(* CODESYS project Vorlage_Visualisierung_Station1.project

Project tree, tasks and I/O mapping:
  SoftSPS : CODESYS Control Win V3 x64, 3S - Smart Software Solutions GmbH, version 3.5.16.40
    application Application
      libraries: Standard, 3.5.15.0 (System)
      task MainTask (cyclic, interval t#15ms, priority 10) calls PLC_PRG
      task VISU_TASK (cyclic, interval 15 ms, priority 0) calls VisuElems.Visu_Prg, vis_Ablauf, vis_Zuweisung
      global variables GVL
      visualisation Visualization
      program PLC_PRG [ST]
      function block FB_Automatik [SFC]: Step4_active, Step5_active, Step7_active, Step8_active, Step10_active, Step9_active, Step12_active, Step6_active, Step14_active, Step13_active, Step17_active, Step18_active, Step19_active, Step24_active, Step25_active, Step22_active, Step23_active
      function block FB_Initialisierung [SFC]: Step0_active, Step1_active, Step2_active, Step3_active, Step4_active, Step5_active, Step11_active, Step7_active, Step8_active, Init_active, Step10_active, Step6_active, Step13_active, Step14_active, Step15_active, Step16_active, Step18_active, Step20_active, Step22_active, Step19_active, Step21_active, Step23_active, Step17_active, Step18_active_0, Step19_active_0, Step20_active_0, Step21_active_0, Step22_active_0, Step23_active_0, Step24_active
  libraries: VisuSymbols, 3.5.10.0 (System)
  text list GlobalTextList
  program vis_Zuweisung [ST]
  data type Flasche
  program vis_Ablauf [ST]
  function block FB_Quit [FBD]
  function block FB_Blink [FBD]
  function block FB_Lamps [ST]
  function block FB_BottleIdentification [ST]
*)

// Flasche
TYPE Flasche :
STRUCT
	Gross		:BOOL;
	Weiss		:BOOL;
	PX			:INT;
	PY			:INT;
	Aktiv		:INT;
	Blockiert	:BOOL;
END_STRUCT
END_TYPE

// SoftSPS/Application/GVL
VAR_GLOBAL
	(*INPUT*)
	i_Abtransport_LT		:BOOL;
	i_Annahme_LT_Eingang	:BOOL;
	i_Annahme_VE_heraus		:BOOL;
	i_Annahme_VE_hinein		:BOOL;
	i_Auto					:BOOL;
	i_BEKenn_LS_mitte		:BOOL;
	i_BEKenn_LS_oben		:BOOL;
	i_BEKenn_LT_unten		:BOOL;
	i_Lager1_LT_Ausgang		:BOOL;
	i_Lager1_LT_Eingang		:BOOL;
	i_Lager1_VE_heraus		:BOOL;
	i_Lager1_VE_hinein		:BOOL;
	i_Lager2_LT_Ausgang		:BOOL;
	i_Lager2_LT_Eingang		:BOOL;
	i_Lager2_VE_heraus		:BOOL;
	i_Lager2_VE_hinein		:BOOL;
	i_Lager2_We_gerade		:BOOL;
	i_Lager2_We_kurve		:BOOL;
	i_Lager3_LT_Ausgang		:BOOL;
	i_Lager3_LT_Eingang		:BOOL;
	i_Lager3_VE_heraus		:BOOL;
	i_Lager3_VE_hinein		:BOOL;
	i_Lager3_We_gerade		:BOOL;
	i_Lager3_We_kurve		:BOOL;
	i_Lager4_LT_Ausgang		:BOOL;
	i_Lager4_LT_Eingang		:BOOL;
	i_Lager4_VE_heraus		:BOOL;
	i_Lager4_VE_hinein		:BOOL;
	i_Lager4_We_gerade		:BOOL;
	i_Lager4_We_kurve		:BOOL;
	i_Notaus				:BOOL;
	i_Quit					:BOOL;
	i_Rueckl_LT_Ausgang		:BOOL;
	i_Rueckl_LT_Eingang		:BOOL;
	i_Rueckl_VE_heraus		:BOOL;
	i_Rueckl_VE_hinein		:BOOL;
	i_Rueckl_We_gerade		:BOOL;
	i_Rueckl_We_kurve		:BOOL;
	i_Schritt				:BOOL;
	i_Weiter				:BOOL;
	(*OUTPUT*)		
	o_Annahme_Band			:BOOL;
	o_Annahme_VE			:BOOL;
	o_Auto					:BOOL;
	o_Fehler				:BOOL;
	o_Lager1_Band			:BOOL;
	o_Lager1_VE				:BOOL;
	o_Lager2_Band			:BOOL;
	o_Lager2_VE				:BOOL;
	o_Lager2_Weiche			:BOOL;
	o_Lager3_Band			:BOOL;
	o_Lager3_VE				:BOOL;
	o_Lager3_Weiche			:BOOL;
	o_Lager4_Band			:BOOL;
	o_Lager4_VE				:BOOL;
	o_Lager4_Weiche			:BOOL;
	o_Rueckl_Band			:BOOL;
	o_Rueckl_VE				:BOOL;
	o_Rueckl_Weiche			:BOOL;
	o_Sammelband_anaus		:BOOL;
	o_Sammelband_Richtung	:BOOL;
	o_Schritt				:BOOL;
	o_Status				:BOOL;
	o_Weichenband			:BOOL;		
END_VAR

// SoftSPS/Application/PLC_PRG
PROGRAM PLC_PRG
VAR
	fb_Quit	:FB_Quit;
	fb_Blink:FB_Blink;
	fb_Lamps:FB_Lamps;
	fb_Automatik: FB_Automatik;
	fb_Initialisierung:FB_Initialisierung;
	m_Idle:					BOOL;
	m_Init:					BOOL;
	m_Automatic:			BOOL;
	m_EmergencyOff:			BOOL;
	m_temp_InitSuccessful:	BOOL;
	m_Fehler:				BOOL;
END_VAR

fb_Quit(i_quittieren:=GVL.i_Quit);

IF NOT GVL.i_Notaus THEN
 m_EmergencyOff := 1;
 m_Idle := 0;
 m_Init := 0;
 m_Automatic := 0;
 m_temp_InitSuccessful:=0;
 
END_IF

IF m_Idle AND GVL.i_Schritt THEN
 m_Init := 1;
 m_Idle := 0;
 m_EmergencyOff :=0;
 m_Automatic :=0;
 fb_Initialisierung(SFCInit:=1);	
END_IF

IF m_Init AND NOT m_temp_InitSuccessful THEN
	fb_Initialisierung(SFCInit:=0);
	m_temp_InitSuccessful:=fb_Initialisierung.o_InitSuccessful;
END_IF

IF m_Init AND m_temp_InitSuccessful AND GVL.i_Auto THEN
 m_Automatic := 1;
 m_EmergencyOff :=0;
 m_Idle :=0;
 m_Init :=0;
END_IF

fb_Lamps(i_Idle:=m_Idle,i_Init:=m_Init,i_EmergencyOff:= m_EmergencyOff,i_Automatic:= m_Automatic,i_EmergencyOffButton:= GVL.i_Notaus,i_InitSuccessful:= m_temp_InitSuccessful,i_Fehler:=m_Fehler);

GVL.o_Status:=fb_Lamps.o_Status;
GVL.o_Fehler:=fb_Lamps.o_Fehler;
GVL.o_Auto:=fb_Lamps.o_Auto;
GVL.o_Schritt:=fb_Lamps.o_Schritt; 

IF m_EmergencyOff AND GVL.i_Notaus AND fb_Quit.o_quittieren THEN
 m_Idle := 1;
 m_EmergencyOff :=0;
 m_Init :=0;
 m_Automatic  :=0; 
 m_temp_InitSuccessful:=0;
END_IF



WHILE m_Automatic AND GVL.i_Notaus DO	
	fb_Automatik(SFCInit:=0);
END_WHILE

IF m_Automatic AND NOT GVL.i_Notaus THEN
	fb_Automatik(SFCInit:=1);
END_IF

END_PROGRAM

// FB_Quit
FUNCTION_BLOCK FB_Quit
VAR_INPUT
	i_quittieren: BOOL;
END_VAR
VAR_OUTPUT
	 o_quittieren: BOOL;
END_VAR
VAR
	f_trig_0: F_TRIG;
	ton_0: TON;
	tp_0: TP;
	tp_1: TP;
	TON_1: TON;
END_VAR

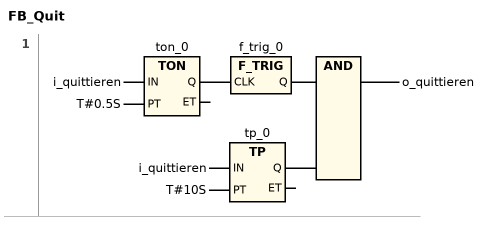
// NETWORK 1
ton_0(IN := i_quittieren, PT := T#0.5S); // TON
f_trig_0(CLK := ton_0.Q); // F_TRIG
tp_0(IN := i_quittieren, PT := T#10S); // TP
o_quittieren := f_trig_0.Q AND tp_0.Q;

END_FUNCTION_BLOCK

// SoftSPS/Application/FB_Initialisierung
FUNCTION_BLOCK FB_Initialisierung
VAR_INPUT
	SFCInit : BOOL;
END_VAR
VAR_OUTPUT
	o_InitSuccessful:BOOL;
END_VAR
VAR
	fb_BottleIdentification :FB_BottleIdentification;
	fb_Ton:Ton;
	h:INT;
	bottleType: INT;
	lagerFrei: BOOL;
	flascheAngekommen: BOOL;
END_VAR

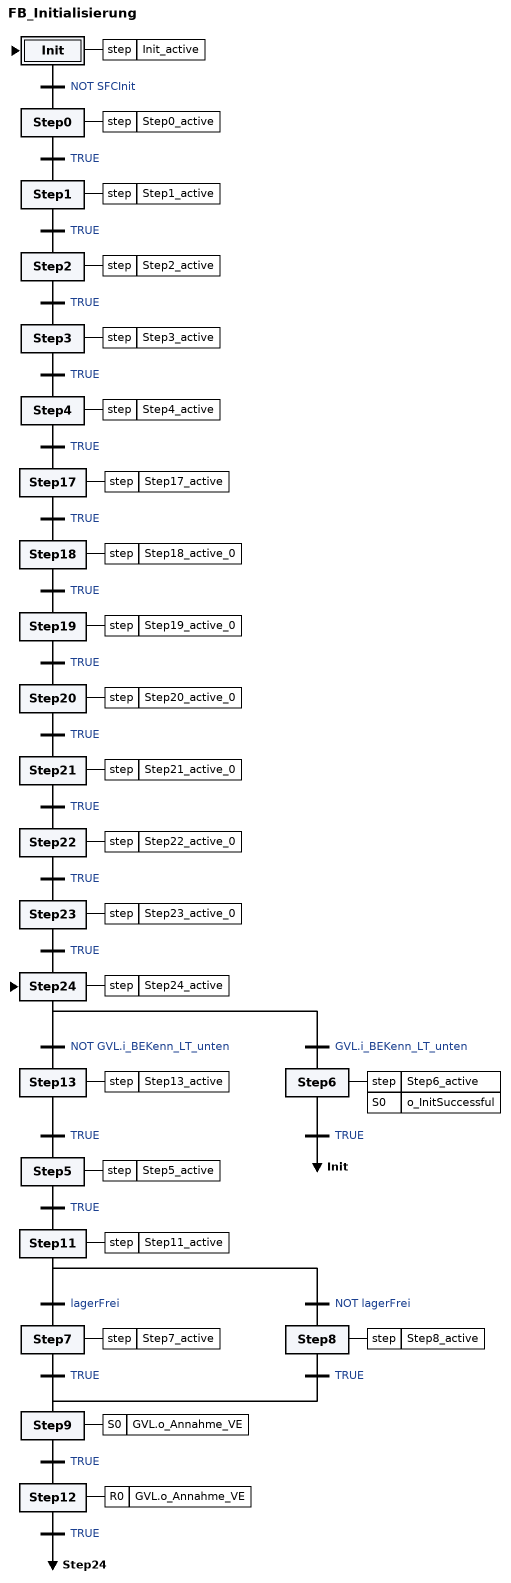
INITIAL_STEP Init:
    Init_active(N);  // step action
END_STEP
TRANSITION FROM Init TO Step0
    := NOT SFCInit;
END_TRANSITION
STEP Step0:
    Step0_active(N);  // step action
END_STEP
TRANSITION FROM Step0 TO Step1
    := TRUE;
END_TRANSITION
STEP Step1:  // min time T#1s
    Step1_active(N);  // step action
END_STEP
TRANSITION FROM Step1 TO Step2
    := TRUE;
END_TRANSITION
STEP Step2:  // min time T#1s
    Step2_active(N);  // step action
END_STEP
TRANSITION FROM Step2 TO Step3
    := TRUE;
END_TRANSITION
STEP Step3:  // min time T#1s
    Step3_active(N);  // step action
END_STEP
TRANSITION FROM Step3 TO Step4
    := TRUE;
END_TRANSITION
STEP Step4:  // min time T#2s
    Step4_active(N);  // step action
END_STEP
TRANSITION FROM Step4 TO Step17
    := TRUE;
END_TRANSITION
STEP Step17:  // min time T#1s
    Step17_active(N);  // step action
END_STEP
TRANSITION FROM Step17 TO Step18
    := TRUE;
END_TRANSITION
STEP Step18:  // min time T#1s
    Step18_active_0(N);  // step action
END_STEP
TRANSITION FROM Step18 TO Step19
    := TRUE;
END_TRANSITION
STEP Step19:  // min time T#1s
    Step19_active_0(N);  // step action
END_STEP
TRANSITION FROM Step19 TO Step20
    := TRUE;
END_TRANSITION
STEP Step20:  // min time T#1s
    Step20_active_0(N);  // step action
END_STEP
TRANSITION FROM Step20 TO Step21
    := TRUE;
END_TRANSITION
STEP Step21:  // min time T#1s
    Step21_active_0(N);  // step action
END_STEP
TRANSITION FROM Step21 TO Step22
    := TRUE;
END_TRANSITION
STEP Step22:  // min time T#1s
    Step22_active_0(N);  // step action
END_STEP
TRANSITION FROM Step22 TO Step23
    := TRUE;
END_TRANSITION
STEP Step23:  // min time T#1s
    Step23_active_0(N);  // step action
END_STEP
TRANSITION FROM Step23 TO Step24
    := TRUE;
END_TRANSITION
STEP Step24:  // min time T#10s
    Step24_active(N);  // step action
END_STEP
TRANSITION FROM Step24 TO Step13
    := NOT GVL.i_BEKenn_LT_unten;
END_TRANSITION
STEP Step13:
    Step13_active(N);  // step action
END_STEP
TRANSITION FROM Step13 TO Step5
    := TRUE;
END_TRANSITION
STEP Step5:
    Step5_active(N);  // step action
END_STEP
TRANSITION FROM Step5 TO Step11
    := TRUE;
END_TRANSITION
STEP Step11:
    Step11_active(N);  // step action
END_STEP
TRANSITION FROM Step11 TO Step7
    := lagerFrei;
END_TRANSITION
STEP Step7:
    Step7_active(N);  // step action
END_STEP
TRANSITION FROM Step7 TO Step9
    := TRUE;
END_TRANSITION
TRANSITION FROM Step11 TO Step8
    := NOT lagerFrei;
END_TRANSITION
STEP Step8:
    Step8_active(N);  // step action
END_STEP
TRANSITION FROM Step8 TO Step9
    := TRUE;
END_TRANSITION
STEP Step9:  // min time T#2s
    GVL.o_Annahme_VE(S0);
END_STEP
TRANSITION FROM Step9 TO Step12
    := TRUE;
END_TRANSITION
STEP Step12:  // min time T#5s
    GVL.o_Annahme_VE(R0);
END_STEP
TRANSITION FROM Step12 TO Step24
    := TRUE;
END_TRANSITION
TRANSITION FROM Step24 TO Step6
    := GVL.i_BEKenn_LT_unten;
END_TRANSITION
STEP Step6:
    Step6_active(N);  // step action
    o_InitSuccessful(S0);
END_STEP
TRANSITION FROM Step6 TO Init
    := TRUE;
END_TRANSITION

ACTION Step0_active:
GVL.o_Annahme_VE:=0;
GVL.o_Lager1_VE:=1;
GVL.o_Lager2_VE:=1;
GVL.o_Lager3_VE:=1;
GVL.o_Lager4_VE:=1;
GVl.o_Rueckl_VE:=1;
GVL.o_Weichenband:=1;
END_ACTION

ACTION Step1_active:
GVL.o_Annahme_Band:=1;
GVL.o_Rueckl_Band:=1;
GVL.o_Rueckl_VE:=1;
END_ACTION

ACTION Step2_active:
GVL.o_Lager3_Band:=1;
GVL.o_Lager4_Band:=1;
END_ACTION

ACTION Step3_active:
GVL.o_Lager1_Band:=1;
GVL.o_Lager2_Band:=1;
END_ACTION

ACTION Step4_active:
GVL.o_Sammelband_anaus:=1;
GVL.o_Sammelband_Richtung:=1;
END_ACTION

ACTION Step5_active:
fb_BottleIdentification(i_LS_Top:=GVL.i_BEKenn_LS_oben, i_LS_Middle:=GVL.i_BEKenn_LS_mitte);
bottleType:=fb_BottleIdentification.o_BottleType;
END_ACTION

ACTION Step11_active:
CASE bottleType OF
	1: 	IF GVL.i_Lager1_LT_Eingang THEN
			lagerFrei:=1;
		ELSE
			lagerFrei:=0;	
		END_IF
	2: 	IF GVL.i_Lager2_LT_Eingang THEN
			lagerFrei:=1;
		ELSE
			lagerFrei:=0;	
		END_IF
	3: 	IF GVL.i_Lager3_LT_Eingang THEN
			lagerFrei:=1;
		ELSE
			lagerFrei:=0;	
		END_IF
	4: 	IF GVL.i_Lager4_LT_Eingang THEN
			lagerFrei:=1;
		ELSE
			lagerFrei:=0;	
		END_IF
END_CASE
END_ACTION

ACTION Step7_active:
CASE bottleType OF
	
	2: GVL.o_Lager2_Weiche:=1;
	3: GVL.o_Lager3_Weiche:=1;	
	4: GVL.o_Lager4_Weiche:=1;	

END_CASE
END_ACTION

ACTION Step8_active:
GVL.o_Rueckl_Weiche:=1;
END_ACTION

ACTION Init_active:
IF SFCInit THEN
	GVL.o_Lager1_Band:=0;
	GVL.o_Lager1_Band:=0;
	GVL.o_Lager1_Band:=0;
	GVL.o_Lager1_Band:=0;
	GVL.o_Annahme_Band:=0;
	GVL.o_Rueckl_Band:=0;
	GVL.o_Weichenband:=0;
	GVL.o_Sammelband_anaus:=0;
	
END_IF
END_ACTION

ACTION Step10_active:

END_ACTION

ACTION Step6_active:
GVL.o_Lager2_Weiche:=0;
GVL.o_Lager3_Weiche:=0;
GVL.o_Lager4_Weiche:=0;
GVL.o_Rueckl_Weiche:=0;

GVL.o_Annahme_Band:=0;
GVL.o_Rueckl_Band:=0;
GVL.o_Lager3_Band:=0;
GVL.o_Lager4_Band:=0;
GVL.o_Lager1_Band:=0;
GVL.o_Lager2_Band:=0;
GVL.o_Sammelband_anaus:=0;
END_ACTION

ACTION Step13_active:
GVL.o_Lager2_Weiche:=0;
GVL.o_Lager3_Weiche:=0;
GVL.o_Lager4_Weiche:=0;
GVL.o_Rueckl_Weiche:=0;
END_ACTION

ACTION Step14_active:
// NETWORK 1
END_ACTION

ACTION Step15_active:
GVL.o_Rueckl_VE:=0;
END_ACTION

ACTION Step16_active:
GVL.o_Rueckl_VE:=1;
END_ACTION

ACTION Step18_active:
GVL.o_Rueckl_VE:=0;
END_ACTION

ACTION Step20_active:

END_ACTION

ACTION Step22_active:
GVL.o_Rueckl_VE:=0;
END_ACTION

ACTION Step19_active:
GVL.o_Rueckl_VE:=1;
END_ACTION

ACTION Step21_active:
GVL.o_Rueckl_VE:=1;
END_ACTION

ACTION Step23_active:
GVL.o_Rueckl_VE:=1;
END_ACTION

ACTION Step17_active:
GVL.o_Rueckl_VE :=0;
END_ACTION

ACTION Step18_active_0:
GVL.o_Rueckl_VE :=1;
END_ACTION

ACTION Step19_active_0:
GVL.o_Rueckl_VE :=0;
END_ACTION

ACTION Step20_active_0:
GVL.o_Rueckl_VE :=1;
END_ACTION

ACTION Step21_active_0:
GVL.o_Rueckl_VE :=0;
END_ACTION

ACTION Step22_active_0:
GVL.o_Rueckl_VE :=1;
END_ACTION

ACTION Step23_active_0:
GVL.o_Rueckl_VE :=0;
END_ACTION

ACTION Step24_active:
GVL.o_Rueckl_VE :=1;
END_ACTION

END_FUNCTION_BLOCK

// FB_BottleIdentification
FUNCTION_BLOCK FB_BottleIdentification
VAR_INPUT
i_LS_Top: BOOL;
i_LS_Middle: BOOL;
END_VAR
VAR_OUTPUT
o_BottleType: INT;
END_VAR
VAR
END_VAR

IF i_LS_Top AND i_LS_Middle THEN
 o_BottleType:=1;
ELSIF NOT i_LS_Top AND i_LS_Middle THEN
 o_BottleType:=2;
ELSIF i_LS_Top AND NOT i_LS_Middle THEN
 o_BottleType:=3;
ELSE
 o_BottleType:=4;
END_IF

END_FUNCTION_BLOCK

// FB_Lamps
FUNCTION_BLOCK FB_Lamps
VAR_INPUT
	 i_Idle: BOOL;
	 i_Init: BOOL;
	 i_Fehler: BOOL;
	 i_EmergencyOff: BOOL;
	 i_Automatic: BOOL;
	 i_EmergencyOffButton: BOOL;
	 i_InitSuccessful: BOOL;
     
END_VAR
VAR_OUTPUT
	 o_Status: BOOL;
     o_Fehler: BOOL;
	 o_Auto: BOOL;
	 o_Schritt: BOOL;
END_VAR
VAR
	fb_Blink: FB_Blink;
END_VAR

IF i_Idle  AND NOT i_Automatic THEN
 fb_Blink(i_BlinkTime:=T#1S);
 o_Status:=fb_Blink.o_Blink;
ELSIF NOT i_Idle  AND i_Automatic THEN
 o_Status:=   1;
 o_Auto:=   1;
 o_Schritt:=   0;
ELSIF i_Init AND NOT i_InitSuccessful THEN
 fb_Blink(i_BlinkTime:=T#500MS);
 o_Status:=     1;
 o_Schritt:=fb_Blink.o_Blink;
 
ELSIF i_Init AND i_InitSuccessful THEN
 o_Status:=   1;
  o_Schritt:=   1;
ELSE
 o_Status:=   0;
 o_Auto:=   0;
 o_Schritt:=   0;
END_IF


IF  i_EmergencyOffButton AND i_EmergencyOff AND NOT i_Fehler THEN
 fb_Blink(i_BlinkTime:=T#167MS);
 o_Fehler:=fb_Blink.o_Blink;
ELSIF i_Fehler OR i_EmergencyOff THEN
 o_Fehler:=   1;
ELSE 
 o_Fehler:=   0;
END_IF

END_FUNCTION_BLOCK

// FB_Blink
FUNCTION_BLOCK FB_Blink
VAR_INPUT
	i_BlinkTime: TIME;
END_VAR
VAR_OUTPUT
	o_Blink: BOOL;
END_VAR
VAR
	ton0: TON;
	ton1: TON;
END_VAR

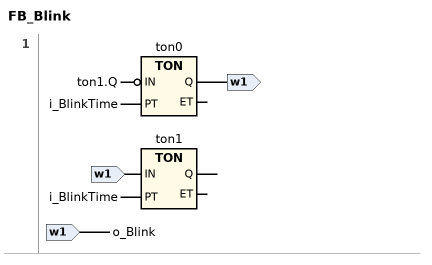
// NETWORK 1
ton0(IN := NOT ton1.Q, PT := i_BlinkTime); // TON
ton1(IN := ton0.Q, PT := i_BlinkTime); // TON
o_Blink := ton0.Q;

END_FUNCTION_BLOCK

// SoftSPS/Application/FB_Automatik
FUNCTION_BLOCK FB_Automatik
VAR_INPUT
	SFCInit : BOOL;
END_VAR
VAR_OUTPUT
END_VAR
VAR
	counter :INT;
	lagerFrei: BOOL;
	fb_BottleIdentification :FB_BottleIdentification;
	bottleType: INT;
	flascheAngekommen: BOOL;
	Timer: BOOL;
	flascheAnLager: BOOL;
END_VAR

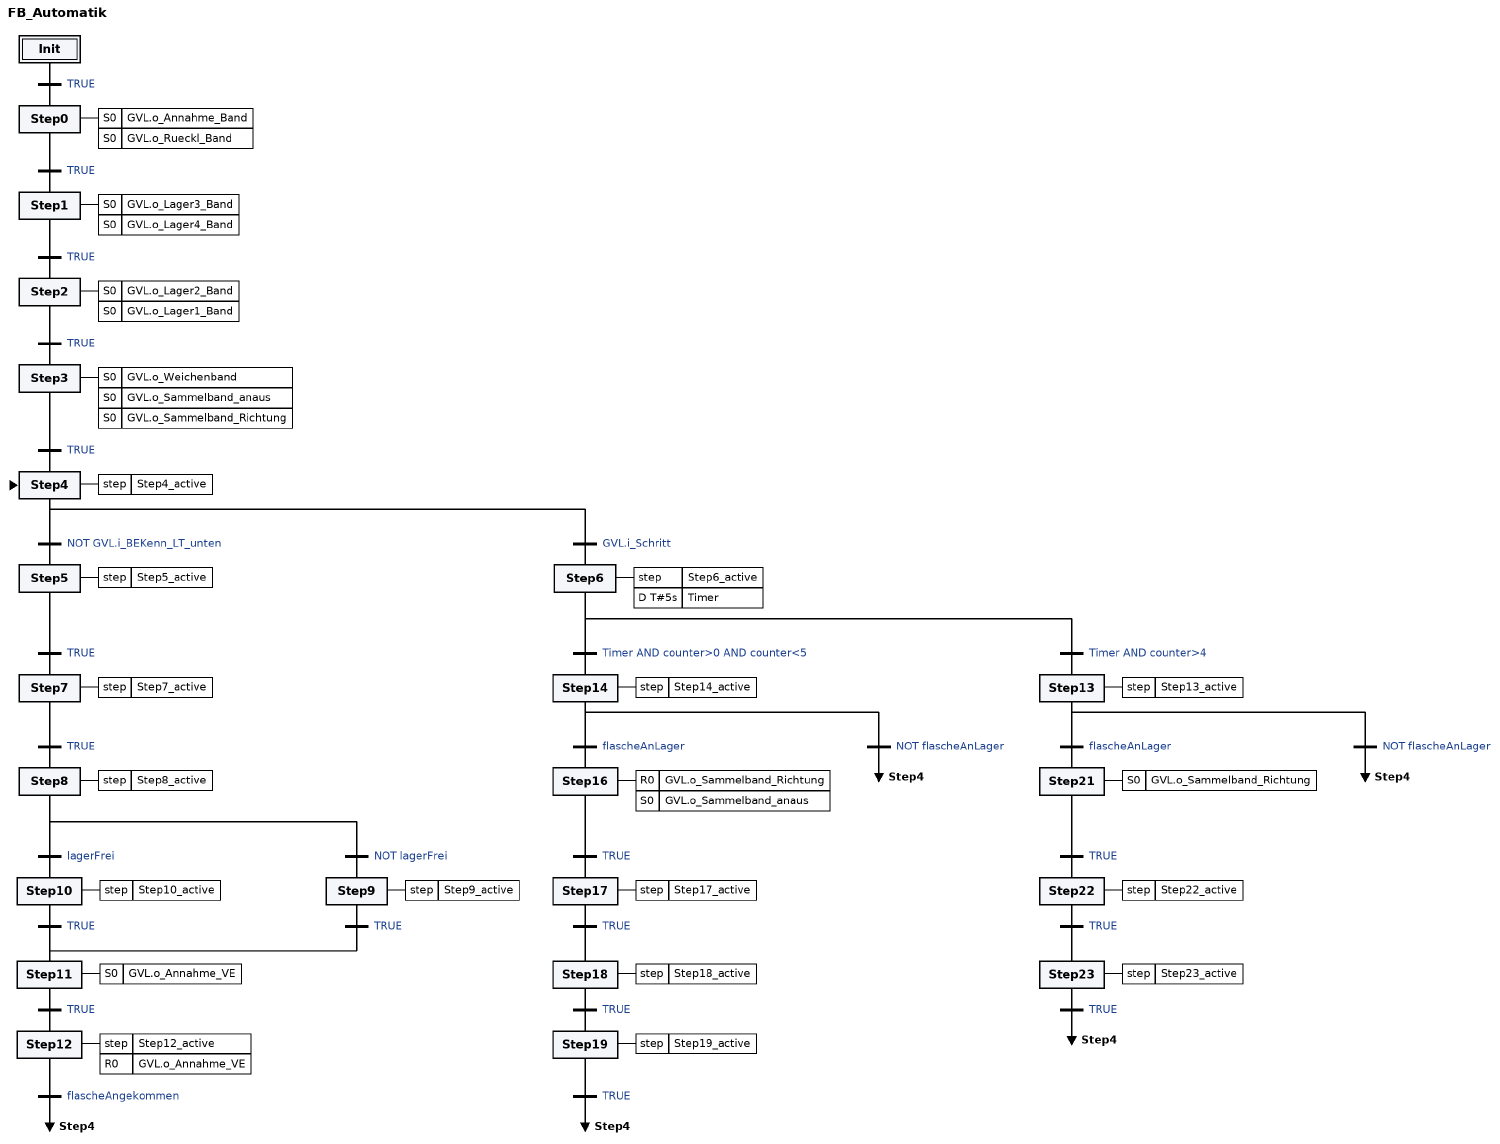
INITIAL_STEP Init:
END_STEP
TRANSITION FROM Init TO Step0
    := TRUE;
END_TRANSITION
STEP Step0:  // min time T#1s
    GVL.o_Annahme_Band(S0);
    GVL.o_Rueckl_Band(S0);
END_STEP
TRANSITION FROM Step0 TO Step1
    := TRUE;
END_TRANSITION
STEP Step1:  // min time T#1s
    GVL.o_Lager3_Band(S0);
    GVL.o_Lager4_Band(S0);
END_STEP
TRANSITION FROM Step1 TO Step2
    := TRUE;
END_TRANSITION
STEP Step2:  // min time T#1s
    GVL.o_Lager2_Band(S0);
    GVL.o_Lager1_Band(S0);
END_STEP
TRANSITION FROM Step2 TO Step3
    := TRUE;
END_TRANSITION
STEP Step3:
    GVL.o_Weichenband(S0);
    GVL.o_Sammelband_anaus(S0);
    GVL.o_Sammelband_Richtung(S0);
END_STEP
TRANSITION FROM Step3 TO Step4
    := TRUE;
END_TRANSITION
STEP Step4:
    Step4_active(N);  // step action
END_STEP
TRANSITION FROM Step4 TO Step5
    := NOT GVL.i_BEKenn_LT_unten;
END_TRANSITION
STEP Step5:
    Step5_active(N);  // step action
END_STEP
TRANSITION FROM Step5 TO Step7
    := TRUE;
END_TRANSITION
STEP Step7:
    Step7_active(N);  // step action
END_STEP
TRANSITION FROM Step7 TO Step8
    := TRUE;
END_TRANSITION
STEP Step8:
    Step8_active(N);  // step action
END_STEP
TRANSITION FROM Step8 TO Step10
    := lagerFrei;
END_TRANSITION
STEP Step10:
    Step10_active(N);  // step action
END_STEP
TRANSITION FROM Step10 TO Step11
    := TRUE;
END_TRANSITION
TRANSITION FROM Step8 TO Step9
    := NOT lagerFrei;
END_TRANSITION
STEP Step9:
    Step9_active(N);  // step action
END_STEP
TRANSITION FROM Step9 TO Step11
    := TRUE;
END_TRANSITION
STEP Step11:  // min time t#2s
    GVL.o_Annahme_VE(S0);
END_STEP
TRANSITION FROM Step11 TO Step12
    := TRUE;
END_TRANSITION
STEP Step12:  // min time T#8s
    Step12_active(N);  // step action
    GVL.o_Annahme_VE(R0);
END_STEP
TRANSITION FROM Step12 TO Step4
    := flascheAngekommen;
END_TRANSITION
TRANSITION FROM Step4 TO Step6
    := GVL.i_Schritt;
END_TRANSITION
STEP Step6:
    Step6_active(N);  // step action
    Timer(D, T#5s);
END_STEP
TRANSITION FROM Step6 TO Step14
    := Timer AND counter>0 AND counter<5;
END_TRANSITION
STEP Step14:
    Step14_active(N);  // step action
END_STEP
TRANSITION FROM Step14 TO Step16
    := flascheAnLager;
END_TRANSITION
STEP Step16:
    GVL.o_Sammelband_Richtung(R0);
    GVL.o_Sammelband_anaus(S0);
END_STEP
TRANSITION FROM Step16 TO Step17
    := TRUE;
END_TRANSITION
STEP Step17:  // min time T#2s
    Step17_active(N);  // step action
END_STEP
TRANSITION FROM Step17 TO Step18
    := TRUE;
END_TRANSITION
STEP Step18:  // min time t#2s
    Step18_active(N);  // step action
END_STEP
TRANSITION FROM Step18 TO Step19
    := TRUE;
END_TRANSITION
STEP Step19:
    Step19_active(N);  // step action
END_STEP
TRANSITION FROM Step19 TO Step4
    := TRUE;
END_TRANSITION
TRANSITION FROM Step14 TO Step4
    := NOT flascheAnLager;
END_TRANSITION
TRANSITION FROM Step6 TO Step13
    := Timer AND counter>4;
END_TRANSITION
STEP Step13:
    Step13_active(N);  // step action
END_STEP
TRANSITION FROM Step13 TO Step21
    := flascheAnLager;
END_TRANSITION
STEP Step21:
    GVL.o_Sammelband_Richtung(S0);
END_STEP
TRANSITION FROM Step21 TO Step22
    := TRUE;
END_TRANSITION
STEP Step22:  // min time t#2s
    Step22_active(N);  // step action
END_STEP
TRANSITION FROM Step22 TO Step23
    := TRUE;
END_TRANSITION
STEP Step23:
    Step23_active(N);  // step action
END_STEP
TRANSITION FROM Step23 TO Step4
    := TRUE;
END_TRANSITION
TRANSITION FROM Step13 TO Step4
    := NOT flascheAnLager;
END_TRANSITION

ACTION Step4_active:
GVL.o_Lager1_VE:=1;
GVL.o_Lager2_VE:=1;
GVL.o_Lager3_VE:=1;
GVL.o_Lager4_VE:=1;

counter:=0;
END_ACTION

ACTION Step5_active:
GVL.o_Lager2_Weiche:=0;
GVL.o_Lager3_Weiche:=0;
GVL.o_Lager4_Weiche:=0;
GVL.o_Rueckl_Weiche:=0;
END_ACTION

ACTION Step7_active:
fb_BottleIdentification(i_LS_Top:=GVL.i_BEKenn_LS_oben, i_LS_Middle:=GVL.i_BEKenn_LS_mitte);
bottleType:=fb_BottleIdentification.o_BottleType;
END_ACTION

ACTION Step8_active:
CASE bottleType OF
	1: 	IF GVL.i_Lager1_LT_Eingang THEN
			lagerFrei:=1;
		ELSE
			lagerFrei:=0;	
		END_IF
	2: 	IF GVL.i_Lager2_LT_Eingang THEN
			lagerFrei:=1;
		ELSE
			lagerFrei:=0;	
		END_IF
	3: 	IF GVL.i_Lager3_LT_Eingang THEN
			lagerFrei:=1;
		ELSE
			lagerFrei:=0;	
		END_IF
	4: 	IF GVL.i_Lager4_LT_Eingang THEN
			lagerFrei:=1;
		ELSE
			lagerFrei:=0;	
		END_IF
END_CASE
END_ACTION

ACTION Step10_active:
CASE bottleType OF
	
	2: GVL.o_Lager2_Weiche:=1;
	3: GVL.o_Lager3_Weiche:=1;	
	4: GVL.o_Lager4_Weiche:=1;	

END_CASE
END_ACTION

ACTION Step9_active:
GVL.o_Rueckl_Weiche:=1;
END_ACTION

ACTION Step12_active:
CASE bottleType OF
	1: 	IF NOT GVL.i_Lager1_LT_Eingang THEN
			flascheAngekommen:=1;
		END_IF
	2: 	IF NOT GVL.i_Lager2_LT_Eingang THEN
			flascheAngekommen:=1;
			
		END_IF
	3:  IF NOT GVL.i_Lager3_LT_Eingang THEN
			flascheAngekommen:=1;
			
		END_IF
	4:  IF NOT GVL.i_Lager4_LT_Eingang THEN
			flascheAngekommen:=1;
			
		END_IF
				
END_CASE
END_ACTION

ACTION Step6_active:
IF i_Schritt THEN
	
	WHILE i_Schritt DO
		counter := counter;
	END_WHILE
	
	counter :=counter+1;
END_IF
END_ACTION

ACTION Step14_active:
CASE counter OF
	
	1: 	IF GVL.i_Lager1_LT_Ausgang THEN
			flascheAnLager :=0;
		ELSE
			flascheAnLager :=1;
		END_IF
	2:  IF GVL.i_Lager2_LT_Ausgang THEN
			flascheAnLager :=0;
		ELSE
			flascheAnLager :=1;			
		END_IF
	3:  IF GVL.i_Lager3_LT_Ausgang THEN
			flascheAnLager :=0;
		ELSE
			flascheAnLager :=1;			
		END_IF
	4:  IF GVL.i_Lager4_LT_Ausgang THEN
			flascheAnLager :=0;
		ELSE
			flascheAnLager :=1;			
		END_IF
		
END_CASE
END_ACTION

ACTION Step13_active:
IF GVL.i_Rueckl_LT_Ausgang THEN
		flascheAnLager :=0;
ELSE
		flascheAnLager :=1;
END_IF
END_ACTION

ACTION Step17_active:
CASE counter OF
	
	1: 	GVL.o_Lager1_VE:=0;
	2:  GVL.o_Lager2_VE:=0;
	3:  GVL.o_Lager3_VE:=0;
	4:  GVL.o_Lager4_VE:=0;
		
END_CASE
END_ACTION

ACTION Step18_active:
CASE counter OF
	
	1: 	GVL.o_Lager1_VE:=1;
	2:  GVL.o_Lager2_VE:=1;
	3:  GVL.o_Lager3_VE:=1;
	4:  GVL.o_Lager4_VE:=1;
		
END_CASE
END_ACTION

ACTION Step19_active:
CASE counter OF
	
	1: 	GVL.o_Lager1_VE:=0;
	2:  GVL.o_Lager2_VE:=0;
	3:  GVL.o_Lager3_VE:=0;
	4:  GVL.o_Lager4_VE:=0;
		
END_CASE
END_ACTION

ACTION Step24_active:
GVL.o_Rueckl_VE :=0;
END_ACTION

ACTION Step25_active:
GVL.o_Rueckl_VE :=1;
END_ACTION

ACTION Step22_active:
GVL.o_Rueckl_VE :=0;
END_ACTION

ACTION Step23_active:
GVL.o_Rueckl_VE :=1;
END_ACTION

END_FUNCTION_BLOCK

// vis_Ablauf
PROGRAM vis_Ablauf
VAR_INPUT 
	Flaschen			:ARRAY [1..50] OF Flasche;
	Taster_Flasche		:ARRAY [1..50] OF BOOL;
	Anlageanaus			:BOOL;
END_VAR

VAR
	i_aktuell		:INT;
	i_Zaehler		:INT;
	i_aktuell_x		:INT;
	i_aktuell_y		:INT;
	Merker_Blockiert	:BOOL;
	
	Pixelpro2Zyklen: INT;
	Zyklus: 		INT;
	initial: 		INT;
	Zykluszaehler: 	INT;
	Merker_AB_LTE	:BOOL;
	Merker_FE_LSU	:BOOL;
	Merker_FE_LSM	:BOOL;
	Merker_FE_LSO	:BOOL;
	Merker_RL_LTE	:BOOL;
	Merker_RL_LTA	:BOOL;
	Merler_L1_LTE	:BOOL;
	Merler_L1_LTA	:BOOL;
	Merler_L2_LTE	:BOOL;
	Merler_L2_LTA	:BOOL;
	Merler_L3_LTE	:BOOL;
	Merler_L3_LTA	:BOOL;
	Merler_L4_LTE	:BOOL;
	Merler_L4_LTA	:BOOL;
	
	i_Zaehler2: 	INT;
	i_Zaehler3: 	INT;
	Startplatz_blockiert: BOOL;
	iInitial: 		INT := 1;
	i_Zaehler4: 	INT;
	Merker_AT_LT: 	BOOL;
	Merker_A5_CB:	BOOL;
	A5_CB_FF	:f_trig;
	A5_CB_RF	:r_trig;
	m_Init_Testcase	:BOOL;
	m_Init_Testcase_einmal :BOOL :=TRUE;
	M_Init_Stellung: BOOL;
	M_Init_Stellung_speicher: BOOL;
	i: INT;
END_VAR

Pixelpro2Zyklen := 1;
Zykluszaehler := Zykluszaehler +1;
IF Zykluszaehler = 1 THEN Zyklus := 1; Zykluszaehler := 0; ELSE Zyklus := 0; END_IF
IF iInitial = 1 THEN
	FOR i_Zaehler4 := 1 TO 50 DO
		IF i_Zaehler4 < 10 THEN Flaschen[i_Zaehler4].Gross := 0; Flaschen[i_Zaehler4].Weiss := 1; END_IF
		IF i_Zaehler4 >= 10 AND i_Zaehler4 < 20 THEN Flaschen[i_Zaehler4].Gross := 1; Flaschen[i_Zaehler4].Weiss := 1; END_IF
		IF i_Zaehler4 >= 20 AND i_Zaehler4 < 30 THEN Flaschen[i_Zaehler4].Gross := 0; Flaschen[i_Zaehler4].Weiss := 0; END_IF
		IF i_Zaehler4 >= 30 AND i_Zaehler4 < 40 THEN Flaschen[i_Zaehler4].Gross := 1; Flaschen[i_Zaehler4].Weiss := 0; END_IF
	END_FOR
	iInitial := 0;
END_IF

IF M_Init_Stellung = TRUE THEN //Einmalige Ausführung
	M_Init_Stellung_speicher:=TRUE;
	
	vis_Zuweisung.vis_o_Lager1_VE			:= TRUE;
	vis_Zuweisung.vis_o_Lager2_VE			:= TRUE;
	vis_Zuweisung.vis_o_Lager3_VE			:= TRUE;
	vis_Zuweisung.vis_o_Lager4_VE			:= TRUE;
	vis_Zuweisung.vis_o_Rueckl_VE			:= TRUE;
	GVL.o_Lager1_VE							:= TRUE;
	GVL.o_Lager2_VE							:= TRUE;
	GVL.o_Lager3_VE							:= TRUE;
	GVL.o_Lager4_VE							:= TRUE;
	GVL.o_Rueckl_VE							:= TRUE;
	GVL.o_Lager2_Weiche 					:= FALSE;
	GVL.o_Lager3_Weiche 					:= FALSE;
	GVL.o_Lager4_Weiche 					:= FALSE;
	GVL.o_Rueckl_Weiche 					:= FALSE;
	
	FOR i := 1 TO 50 DO
		Flaschen[i].Aktiv := 0;
		Flaschen[i].PX := 0;
		Flaschen[i].PY := 0 ;
	END_FOR
	
END_IF

IF M_Init_Stellung_speicher = TRUE THEN //Dauerhafte Ausführung bis Initialisierte Stellung eingenommen übernimmt
	
	IF TRUE THEN
			M_Init_Stellung_speicher := FALSE;
	END_IF
END_IF


IF m_Init_Testcase_einmal = TRUE AND m_Init_Testcase = TRUE THEN
	Flaschen[5].Aktiv := 1;
	Flaschen[5].PX := Flaschen[5].PX + 50;
	Flaschen[5].PY := Flaschen[5].PY ;
	Flaschen[11].Aktiv := 1;
	Flaschen[11].PX := Flaschen[11].PX + 350;
	Flaschen[11].PY := Flaschen[11].PY -90;
	Flaschen[14].Aktiv := 1;
	Flaschen[14].PX := Flaschen[14].PX + 30;
	Flaschen[14].PY := Flaschen[14].PY -390;
	Flaschen[23].Aktiv := 1;
	Flaschen[23].PX := Flaschen[23].PX + 190;
	Flaschen[23].PY := Flaschen[23].PY -90;
	Flaschen[36].Aktiv := 1;
	Flaschen[36].PX := Flaschen[36].PX + 580;
	Flaschen[36].PY := Flaschen[36].PY -200;
	GVL.o_Lager2_Weiche := TRUE;
	vis_Zuweisung.Lager2_Weiche_rot := -55;
	
	
	
	m_Init_Testcase_einmal := FALSE;
END_IF

  
FOR i_Zaehler3 := 1 TO 50 DO
	IF Flaschen[i_Zaehler3].PX <= 50 AND Flaschen[i_Zaehler3].PY = 0 AND Flaschen[i_Zaehler3].Aktiv = 1 THEN Startplatz_blockiert := 1; i_Zaehler3 := 51;
	ELSIF  Merker_A5_CB AND Flaschen[i_Zaehler3].PX <= 350 AND Flaschen[i_Zaehler3].PY = 0 AND Flaschen[i_Zaehler3].Aktiv = 1 THEN Startplatz_blockiert := 1; i_Zaehler3 := 51;
	ELSE Startplatz_blockiert := 0;
	END_IF
END_FOR


FOR i_Zaehler := 1 TO 50 DO
	
IF Taster_Flasche[i_Zaehler] = 1 AND Startplatz_blockiert = 0  THEN Flaschen[i_Zaehler].Aktiv := 1; END_IF

i_aktuell := i_Zaehler;
IF Flaschen[i_aktuell].Aktiv = 1 THEN
	
	i_aktuell_x := Flaschen[i_aktuell].PX;
	i_aktuell_y := Flaschen[i_aktuell].PY;
	

IF Flaschen[i_aktuell].Blockiert = 0 THEN
// Fahren
	
	// Fahren auf Annahmeband
		IF vis_Zuweisung.vis_o_Annahme_Band = 1 AND i_aktuell_y = 0 AND i_aktuell_x >= 0 AND i_aktuell_x < 580 THEN
			i_aktuell_x := i_aktuell_x +  Zyklus*Pixelpro2Zyklen; 
		END_IF
			
	// Fahren auf Rücklaufband
		IF vis_Zuweisung.vis_o_Rueckl_Band = 1 AND i_aktuell_y = -90 AND
		((i_aktuell_x = 580 AND vis_Zuweisung.vis_i_Rueckl_We_kurve = 1) OR (i_aktuell_x > 30 AND i_aktuell_x < 580)) THEN
			i_aktuell_x := i_aktuell_x -  Zyklus*Pixelpro2Zyklen; 
		END_IF
		
	// Fahren in Lager 4
		IF vis_Zuweisung.vis_o_Lager4_Band = 1 AND i_aktuell_y = -190 AND
		((i_aktuell_x = 580 AND vis_Zuweisung.vis_i_Lager4_We_kurve = 1 ) OR (i_aktuell_x > 30 AND i_aktuell_x < 580)) THEN
			i_aktuell_x := i_aktuell_x -  Zyklus*Pixelpro2Zyklen; 
		END_IF
		
	// Fahren in Lager 3
		IF vis_Zuweisung.vis_o_Lager3_Band = 1 AND i_aktuell_y = -290 AND
		((i_aktuell_x = 580 AND vis_Zuweisung.vis_i_Lager3_We_kurve = 1) OR (i_aktuell_x > 30 AND i_aktuell_x < 580)) THEN
			i_aktuell_x := i_aktuell_x -  Zyklus*Pixelpro2Zyklen; 
		END_IF
		
	// Fahren in Lager 2
		IF vis_Zuweisung.vis_o_Lager2_Band = 1 AND i_aktuell_y = -390 AND
		((i_aktuell_x = 580 AND vis_Zuweisung.vis_i_Lager2_We_kurve = 1) OR (i_aktuell_x > 30 AND i_aktuell_x < 580)) THEN
			i_aktuell_x := i_aktuell_x -  Zyklus*Pixelpro2Zyklen; 
		END_IF
		
	// Fahren in Lager 1
		IF vis_Zuweisung.vis_o_Lager1_Band = 1 AND i_aktuell_y = -490 AND i_aktuell_x >= -100 AND i_aktuell_x < 581 THEN
			i_aktuell_x := i_aktuell_x -  Zyklus*Pixelpro2Zyklen; 
		END_IF
		
	// Fahren auf Weichenband
		IF vis_Zuweisung.vis_o_Weichenband = 1 AND i_aktuell_x = 580 AND i_aktuell_y <= 0 AND i_aktuell_y > -490 THEN
			i_aktuell_y := i_aktuell_y -  Zyklus*Pixelpro2Zyklen; 
		END_IF
		
	// Fahren auf Sammelband
		IF vis_Zuweisung.vis_o_Sammelband_anaus = 1 AND i_aktuell_x = 30 AND i_aktuell_y < 0 AND i_aktuell_y > -490 THEN
		IF vis_Zuweisung.vis_o_Sammelband_Richtung = 1 THEN i_aktuell_y := i_aktuell_y +  Zyklus*Pixelpro2Zyklen; END_IF
		IF vis_Zuweisung.vis_o_Sammelband_Richtung = 0 THEN i_aktuell_y := i_aktuell_y -  Zyklus*Pixelpro2Zyklen; END_IF
		END_IF
	
			
		
END_IF

		
// Blockieren durch Weichen und Vereinzeler

		Merker_Blockiert := 0;
// Weichen auf Weichenband
	
	// Weiche Rücklauf
		IF i_aktuell_x = 580 AND i_aktuell_y = -90 AND vis_Zuweisung.vis_i_Rueckl_We_kurve = 1 AND vis_Zuweisung.vis_o_Rueckl_Band = 0 THEN 
		Flaschen[i_aktuell].Blockiert := 1; Merker_Blockiert := 1;
		ELSIF i_aktuell_x = 580 AND i_aktuell_y = -90 AND (vis_Zuweisung.vis_i_Rueckl_We_gerade = 1 OR vis_Zuweisung.vis_o_Rueckl_Band = 1) THEN Flaschen[i_aktuell].Blockiert := 0; 
		END_IF
		
	// Weiche Lager 4
		IF i_aktuell_x = 580 AND i_aktuell_y = -190 AND vis_Zuweisung.vis_i_Lager4_We_kurve = 1 AND vis_Zuweisung.vis_o_Lager4_Band = 0 THEN 
		Flaschen[i_aktuell].Blockiert := 1; Merker_Blockiert := 1;
		ELSIF i_aktuell_x = 580 AND i_aktuell_y = -190 AND (vis_Zuweisung.vis_i_Lager4_We_gerade = 1 OR vis_Zuweisung.vis_o_Lager4_Band = 1) THEN Flaschen[i_aktuell].Blockiert := 0; 
		END_IF
		
	// Weiche Lager 3
		IF i_aktuell_x = 580 AND i_aktuell_y = -290 AND vis_Zuweisung.vis_i_Lager3_We_kurve = 1 AND vis_Zuweisung.vis_o_Lager3_Band = 0 THEN 
		Flaschen[i_aktuell].Blockiert := 1; Merker_Blockiert := 1;
		ELSIF i_aktuell_x = 580 AND i_aktuell_y = -290 AND (vis_Zuweisung.vis_i_Lager3_We_gerade = 1 OR vis_Zuweisung.vis_o_Lager3_Band = 1)THEN Flaschen[i_aktuell].Blockiert := 0; 
		END_IF
		
	// Weiche Lager 2
		IF i_aktuell_x = 580 AND i_aktuell_y = -390 AND vis_Zuweisung.vis_i_Lager2_We_kurve = 1 AND vis_Zuweisung.vis_o_Lager2_Band = 0 THEN 
		Flaschen[i_aktuell].Blockiert := 1; Merker_Blockiert := 1;
		ELSIF i_aktuell_x = 580 AND i_aktuell_y = -390 AND (vis_Zuweisung.vis_i_Lager2_We_gerade = 1 OR vis_Zuweisung.vis_o_Lager2_Band = 1)THEN Flaschen[i_aktuell].Blockiert := 0; 
		END_IF
			
	// Vereinzeler Annahmeband
		IF i_aktuell_x = 501 AND i_aktuell_y = 0 AND vis_Zuweisung.vis_i_Annahme_VE_hinein = 1 THEN 
		Flaschen[i_aktuell].Blockiert := 1; Merker_Blockiert := 1;
		ELSIF i_aktuell_x = 501 AND i_aktuell_y = 0 AND vis_Zuweisung.vis_i_Annahme_VE_heraus = 1 THEN Flaschen[i_aktuell].Blockiert := 0; 
		END_IF
		
		IF i_aktuell_x = 462 AND i_aktuell_y = 0 AND vis_Zuweisung.vis_i_Annahme_VE_heraus = 1 THEN 
		Flaschen[i_aktuell].Blockiert := 1; Merker_Blockiert := 1;
		ELSIF i_aktuell_x = 462 AND i_aktuell_y = 0 AND vis_Zuweisung.vis_i_Annahme_VE_hinein = 1 THEN Flaschen[i_aktuell].Blockiert := 0;
		END_IF
	
	// Vereinzeler Rücklaufband
		IF i_aktuell_x = 100 AND i_aktuell_y = -90 AND vis_Zuweisung.vis_i_Rueckl_VE_hinein = 1 THEN 
		Flaschen[i_aktuell].Blockiert := 1; Merker_Blockiert := 1;
		ELSIF i_aktuell_x = 100 AND i_aktuell_y = -90 AND vis_Zuweisung.vis_i_Rueckl_VE_heraus = 1 THEN Flaschen[i_aktuell].Blockiert := 0; 
		END_IF
		
		IF i_aktuell_x = 140 AND i_aktuell_y = -90 AND vis_Zuweisung.vis_i_Rueckl_VE_heraus = 1 THEN 
		Flaschen[i_aktuell].Blockiert := 1; Merker_Blockiert := 1;
		ELSIF i_aktuell_x = 140 AND i_aktuell_y = -90 AND vis_Zuweisung.vis_i_Rueckl_VE_hinein = 1 THEN Flaschen[i_aktuell].Blockiert := 0;
		END_IF
		
	// Vereinzeler Lager 4
		IF i_aktuell_x = 100 AND i_aktuell_y = -190 AND vis_Zuweisung.vis_i_Lager4_VE_hinein = 1 THEN 
		Flaschen[i_aktuell].Blockiert := 1; Merker_Blockiert := 1;
		ELSIF i_aktuell_x = 100 AND i_aktuell_y = -190 AND vis_Zuweisung.vis_i_Lager4_VE_heraus = 1 THEN Flaschen[i_aktuell].Blockiert := 0; 
		END_IF
		
		IF i_aktuell_x = 140 AND i_aktuell_y = -190 AND vis_Zuweisung.vis_i_Lager4_VE_heraus = 1 THEN 
		Flaschen[i_aktuell].Blockiert := 1; Merker_Blockiert := 1;
		ELSIF i_aktuell_x = 140 AND i_aktuell_y = -190 AND vis_Zuweisung.vis_i_Lager4_VE_hinein = 1 THEN Flaschen[i_aktuell].Blockiert := 0;
		END_IF
	
	// Vereinzeler Lager 3
		IF i_aktuell_x = 100 AND i_aktuell_y = -290 AND vis_Zuweisung.vis_i_Lager3_VE_hinein = 1 THEN 
		Flaschen[i_aktuell].Blockiert := 1; Merker_Blockiert := 1;
		ELSIF i_aktuell_x = 100 AND i_aktuell_y = -290 AND vis_Zuweisung.vis_i_Lager3_VE_heraus = 1 THEN Flaschen[i_aktuell].Blockiert := 0; 
		END_IF
		
		IF i_aktuell_x = 140 AND i_aktuell_y = -290 AND vis_Zuweisung.vis_i_Lager3_VE_heraus = 1 THEN 
		Flaschen[i_aktuell].Blockiert := 1; Merker_Blockiert := 1;
		ELSIF i_aktuell_x = 140 AND i_aktuell_y = -290 AND vis_Zuweisung.vis_i_Lager3_VE_hinein = 1 THEN Flaschen[i_aktuell].Blockiert := 0;
		END_IF
		
	// Vereinzeler Lager 2
		IF i_aktuell_x = 100 AND i_aktuell_y = -390 AND vis_Zuweisung.vis_i_Lager2_VE_hinein = 1 THEN 
		Flaschen[i_aktuell].Blockiert := 1; Merker_Blockiert := 1;
		ELSIF i_aktuell_x = 100 AND i_aktuell_y = -390 AND vis_Zuweisung.vis_i_Lager2_VE_heraus = 1 THEN Flaschen[i_aktuell].Blockiert := 0; 
		END_IF
		
		IF i_aktuell_x = 140 AND i_aktuell_y = -390 AND vis_Zuweisung.vis_i_Lager2_VE_heraus = 1 THEN 
		Flaschen[i_aktuell].Blockiert := 1; Merker_Blockiert := 1;
		ELSIF i_aktuell_x = 140 AND i_aktuell_y = -390 AND vis_Zuweisung.vis_i_Lager2_VE_hinein = 1 THEN Flaschen[i_aktuell].Blockiert := 0;
		END_IF
	
	// Vereinzeler Lager 1
		IF i_aktuell_x = 100 AND i_aktuell_y = -490 AND vis_Zuweisung.vis_i_Lager1_VE_hinein = 1 THEN 
		Flaschen[i_aktuell].Blockiert := 1; Merker_Blockiert := 1;
		ELSIF i_aktuell_x = 100 AND i_aktuell_y = -490 AND vis_Zuweisung.vis_i_Lager1_VE_heraus = 1 THEN Flaschen[i_aktuell].Blockiert := 0; 
		END_IF
		
		IF i_aktuell_x = 140 AND i_aktuell_y = -490 AND vis_Zuweisung.vis_i_Lager1_VE_heraus = 1 THEN 
		Flaschen[i_aktuell].Blockiert := 1; Merker_Blockiert := 1;
		ELSIF i_aktuell_x = 140 AND i_aktuell_y = -490 AND vis_Zuweisung.vis_i_Lager1_VE_hinein = 1 THEN Flaschen[i_aktuell].Blockiert := 0;
		END_IF
		
// Blockieren durch andere Flaschen
	FOR i_Zaehler2 := 1 TO 50 DO
		
	// Auf Annahmeband
		IF i_aktuell_x >= 0 AND i_aktuell_x < 570 AND i_aktuell_y = 0 AND Merker_Blockiert = 0 THEN
			IF (i_aktuell_x = Flaschen[i_Zaehler2].PX - 50) AND (Flaschen[i_Zaehler2].PY = 0) AND Flaschen[i_Zaehler2].Aktiv = 1 THEN Flaschen[i_aktuell].Blockiert := 1; i_Zaehler2 := 51;
			ELSE Flaschen[i_aktuell].Blockiert := 0;
			END_IF
		END_IF
		
	// Auf Weichenband
		IF i_aktuell_x >= -490 AND i_aktuell_y < 0 AND i_aktuell_x < 531 AND Merker_Blockiert = 0 THEN
			IF (i_aktuell_y = Flaschen[i_Zaehler2].PY + 50) AND (Flaschen[i_Zaehler2].PX = 580) AND Flaschen[i_Zaehler2].Aktiv = 1 THEN Flaschen[i_aktuell].Blockiert := 1; i_Zaehler2 := 51;
			ELSE Flaschen[i_aktuell].Blockiert := 0;
			END_IF
		END_IF
		
	// Auf Rücklaufband
		IF i_aktuell_x >= 30 AND i_aktuell_x < 570 AND i_aktuell_y = -90 AND Merker_Blockiert = 0 THEN
			IF (i_aktuell_x = Flaschen[i_Zaehler2].PX + 50) AND (Flaschen[i_Zaehler2].PY = -90) AND Flaschen[i_Zaehler2].Aktiv = 1 THEN Flaschen[i_aktuell].Blockiert := 1; i_Zaehler2 := 51;
			ELSE Flaschen[i_aktuell].Blockiert := 0;
			END_IF
		END_IF
		
	// In Lager 4
		IF i_aktuell_x >= 30 AND i_aktuell_x < 570 AND i_aktuell_y = -190 AND Merker_Blockiert = 0 THEN
			IF (i_aktuell_x = Flaschen[i_Zaehler2].PX + 50) AND (Flaschen[i_Zaehler2].PY = -190) AND Flaschen[i_Zaehler2].Aktiv = 1 THEN Flaschen[i_aktuell].Blockiert := 1; i_Zaehler2 := 51;
			ELSE Flaschen[i_aktuell].Blockiert := 0;
			END_IF
		END_IF
	
	// In Lager 3
		IF i_aktuell_x >= 30 AND i_aktuell_x < 570 AND i_aktuell_y = -290 AND Merker_Blockiert = 0 THEN
			IF (i_aktuell_x = Flaschen[i_Zaehler2].PX + 50) AND (Flaschen[i_Zaehler2].PY = -290) AND Flaschen[i_Zaehler2].Aktiv = 1 THEN Flaschen[i_aktuell].Blockiert := 1; i_Zaehler2 := 51;
			ELSE Flaschen[i_aktuell].Blockiert := 0;
			END_IF
		END_IF
		
	// In Lager 2
		IF i_aktuell_x >= 30 AND i_aktuell_x < 570 AND i_aktuell_y = -390 AND Merker_Blockiert = 0 THEN
			IF (i_aktuell_x = Flaschen[i_Zaehler2].PX + 50) AND (Flaschen[i_Zaehler2].PY = -390) AND Flaschen[i_Zaehler2].Aktiv = 1 THEN Flaschen[i_aktuell].Blockiert := 1; i_Zaehler2 := 51;
			ELSE Flaschen[i_aktuell].Blockiert := 0;
			END_IF
		END_IF
		
	// in Lager 1
		IF i_aktuell_x >= -100 AND i_aktuell_x < 581 AND i_aktuell_y = -490 AND Merker_Blockiert = 0 THEN
			IF (i_aktuell_x = Flaschen[i_Zaehler2].PX + 50) AND (Flaschen[i_Zaehler2].PY = -490) AND Flaschen[i_Zaehler2].Aktiv = 1 THEN Flaschen[i_aktuell].Blockiert := 1; i_Zaehler2 := 51;
			ELSE Flaschen[i_aktuell].Blockiert := 0;
			END_IF
		END_IF
		
	END_FOR	
// Flaschen zurücksetzen wenn Ausgang erreicht
	IF i_aktuell_x = -98 AND i_aktuell_y = -490 THEN
		i_aktuell_x := 0;
		i_aktuell_y := 0;
		Flaschen[i_aktuell].Aktiv := 0;
	END_IF 	
	
	
// Schreiben der Position		
	Flaschen[i_aktuell].PX := i_aktuell_x;
	Flaschen[i_aktuell].PY := i_aktuell_y;
	
END_IF	
END_FOR

// Weichenmanagement

IF vis_Zuweisung.vis_o_Annahme_VE = 0 THEN 
	vis_Zuweisung.Annahme_VE_rot := 38; vis_Zuweisung.vis_i_Annahme_VE_heraus := 1; vis_Zuweisung.vis_i_Annahme_VE_hinein := 0;
	ELSE vis_Zuweisung.Annahme_VE_rot := 0; vis_Zuweisung.vis_i_Annahme_VE_heraus := 0;  vis_Zuweisung.vis_i_Annahme_VE_hinein := 1;
END_IF

IF vis_Zuweisung.vis_o_Lager1_VE = 1 THEN 
	vis_Zuweisung.Lager1_VE_rot := 30; vis_Zuweisung.vis_i_Lager1_VE_heraus := 1; vis_Zuweisung.vis_i_Lager1_VE_hinein := 0;
	ELSE vis_Zuweisung.Lager1_VE_rot := 0; vis_Zuweisung.vis_i_Lager1_VE_heraus := 0;  vis_Zuweisung.vis_i_Lager1_VE_hinein := 1;
END_IF

IF vis_Zuweisung.vis_o_Lager2_VE = 1 THEN 
	vis_Zuweisung.Lager2_VE_rot := 30; vis_Zuweisung.vis_i_Lager2_VE_heraus := 1; vis_Zuweisung.vis_i_Lager2_VE_hinein := 0;
	ELSE vis_Zuweisung.Lager2_VE_rot := 0; vis_Zuweisung.vis_i_Lager2_VE_heraus := 0;  vis_Zuweisung.vis_i_Lager2_VE_hinein := 1;
END_IF

IF vis_Zuweisung.vis_o_Lager3_VE = 1 THEN 
	vis_Zuweisung.Lager3_VE_rot := 30; vis_Zuweisung.vis_i_Lager3_VE_heraus := 1; vis_Zuweisung.vis_i_Lager3_VE_hinein := 0;
	ELSE vis_Zuweisung.Lager3_VE_rot := 0; vis_Zuweisung.vis_i_Lager3_VE_heraus := 0;  vis_Zuweisung.vis_i_Lager3_VE_hinein := 1;
END_IF

IF vis_Zuweisung.vis_o_Lager4_VE = 1 THEN 
	vis_Zuweisung.Lager4_VE_rot := 30; vis_Zuweisung.vis_i_Lager4_VE_heraus := 1; vis_Zuweisung.vis_i_Lager4_VE_hinein := 0;
	ELSE vis_Zuweisung.Lager4_VE_rot := 0; vis_Zuweisung.vis_i_Lager4_VE_heraus := 0;  vis_Zuweisung.vis_i_Lager4_VE_hinein := 1;
END_IF

IF vis_Zuweisung.vis_o_Rueckl_VE = 1 THEN 
	vis_Zuweisung.Rueckl_VE_rot := 30; vis_Zuweisung.vis_i_Rueckl_VE_heraus := 1; vis_Zuweisung.vis_i_Rueckl_VE_hinein := 0;
	ELSE vis_Zuweisung.Rueckl_VE_rot := 0; vis_Zuweisung.vis_i_Rueckl_VE_heraus := 0;  vis_Zuweisung.vis_i_Rueckl_VE_hinein := 1;
END_IF

IF vis_Zuweisung.vis_o_Lager2_Weiche = 1 THEN 
	vis_Zuweisung.Lager2_Weiche_rot := -55; vis_Zuweisung.vis_i_Lager2_We_kurve := 1; vis_Zuweisung.vis_i_Lager2_We_gerade := 0;
	ELSE vis_Zuweisung.Lager2_Weiche_rot := 0; vis_Zuweisung.vis_i_Lager2_We_kurve := 0;  vis_Zuweisung.vis_i_Lager2_We_gerade := 1;
END_IF

IF vis_Zuweisung.vis_o_Lager3_Weiche = 1 THEN 
	vis_Zuweisung.Lager3_Weiche_rot := -55; vis_Zuweisung.vis_i_Lager3_We_kurve := 1; vis_Zuweisung.vis_i_Lager3_We_gerade := 0;
	ELSE vis_Zuweisung.Lager3_Weiche_rot := 0; vis_Zuweisung.vis_i_Lager3_We_kurve := 0;  vis_Zuweisung.vis_i_Lager3_We_gerade := 1;
END_IF

IF vis_Zuweisung.vis_o_Lager4_Weiche = 1 THEN 
	vis_Zuweisung.Lager4_Weiche_rot := -55; vis_Zuweisung.vis_i_Lager4_We_kurve := 1; vis_Zuweisung.vis_i_Lager4_We_gerade := 0;
	ELSE vis_Zuweisung.Lager4_Weiche_rot := 0; vis_Zuweisung.vis_i_Lager4_We_kurve := 0;  vis_Zuweisung.vis_i_Lager4_We_gerade := 1;
END_IF

IF vis_Zuweisung.vis_o_Rueckl_Weiche = 1 THEN 
	vis_Zuweisung.Rueckl_Weiche_rot := -55; vis_Zuweisung.vis_i_Rueckl_We_kurve := 1; vis_Zuweisung.vis_i_Rueckl_We_gerade := 0;
	ELSE vis_Zuweisung.Rueckl_Weiche_rot := 0; vis_Zuweisung.vis_i_Rueckl_We_kurve := 0;  vis_Zuweisung.vis_i_Rueckl_We_gerade := 1;
END_IF

// Sensorenmanagement
	
	Merker_AT_LT	:= 0;
	Merker_AB_LTE	:= 0;
	Merker_FE_LSU	:= 0;
	Merker_FE_LSM	:= 0;
	Merker_FE_LSO	:= 0;
	Merker_RL_LTE	:= 0;
	Merker_RL_LTA	:= 0;
	Merler_L1_LTE	:= 0;
	Merler_L1_LTA	:= 0;
	Merler_L2_LTE	:= 0;
	Merler_L2_LTA	:= 0;
	Merler_L3_LTE	:= 0;
	Merler_L3_LTA	:= 0;
	Merler_L4_LTE	:= 0;
	Merler_L4_LTA	:= 0;
	
FOR i_Zaehler := 1 TO 50 DO
	
	// Abtransport LT
	IF Merker_AT_LT = 0 THEN
	IF Flaschen[i_Zaehler].PX > -60 AND Flaschen[i_Zaehler].PX < -20 AND Flaschen[i_Zaehler].PY = -490 
		THEN vis_Zuweisung.vis_i_Abtransport_LT := 0; Merker_AT_LT := 1;
		ELSE vis_Zuweisung.vis_i_Abtransport_LT := 1;
	END_IF
	END_IF

	// Annahmeband LT Eingang
	IF Merker_AB_LTE = 0 THEN
	IF Flaschen[i_Zaehler].PX > 76 AND Flaschen[i_Zaehler].PX < 104 AND Flaschen[i_Zaehler].PY = 0 
		THEN vis_Zuweisung.vis_i_Annahme_LT_Eingang := 0; Merker_AB_LTE := 1;
		ELSE vis_Zuweisung.vis_i_Annahme_LT_Eingang := 1;
	END_IF
	END_IF
	
	// Flaschenerkennung
	IF Merker_FE_LSU = 0 THEN
	IF Flaschen[i_Zaehler].PX > 440 AND Flaschen[i_Zaehler].PX < 472 AND Flaschen[i_Zaehler].PY = 0
 	THEN vis_Zuweisung.vis_i_BEKenn_LS_unten := 0; Merker_FE_LSU := 1;
		ELSE vis_Zuweisung.vis_i_BEKenn_LS_unten := 1;
	END_IF
	END_IF
	
	IF Merker_FE_LSM = 0 THEN
	IF (((Flaschen[i_Zaehler].PX > 430 AND Flaschen[i_Zaehler].PX < 436) OR (Flaschen[i_Zaehler].PX > 465
		AND Flaschen[i_Zaehler].PX < 471)) OR (Flaschen[i_Zaehler].PX > 435 AND Flaschen[i_Zaehler].PX < 465 AND Flaschen[i_Zaehler].Weiss = 0)) AND Flaschen[i_Zaehler].PY = 0 
		THEN vis_Zuweisung.vis_i_BEKenn_LS_mitte := 1; Merker_FE_LSM := 1;
		ELSE vis_Zuweisung.vis_i_BEKenn_LS_mitte := 0;
	END_IF
	END_IF
	
	IF Merker_FE_LSO = 0 THEN
	IF Flaschen[i_Zaehler].PX > 438 AND Flaschen[i_Zaehler].PX < 478 AND Flaschen[i_Zaehler].PY = 0 AND Flaschen[i_Zaehler].Gross = 0 
		THEN vis_Zuweisung.vis_i_BEKenn_LS_oben := 1; Merker_FE_LSO := 1;
		ELSE vis_Zuweisung.vis_i_BEKenn_LS_oben := 0;
	END_IF
	END_IF
	
	//Rücklauf LT_Eingang
	IF Merker_RL_LTE = 0 THEN
	IF Flaschen[i_Zaehler].PY = -90 AND Flaschen[i_Zaehler].PX > 485 AND Flaschen[i_Zaehler].PX < 495 
		THEN vis_Zuweisung.vis_i_Rueckl_LT_Eingang := 0; Merker_RL_LTE := 1;
		ELSE vis_Zuweisung.vis_i_Rueckl_LT_Eingang := 1;
	END_IF
	END_IF
	
	// Lager 4 LT_Eingang
	IF Merler_L4_LTE = 0 THEN
	IF Flaschen[i_Zaehler].PY = -190 AND Flaschen[i_Zaehler].PX > 485 AND Flaschen[i_Zaehler].PX < 495
		THEN vis_Zuweisung.vis_i_Lager4_LT_Eingang := 0; Merler_L4_LTE := 1;
		ELSE vis_Zuweisung.vis_i_Lager4_LT_Eingang := 1;
	END_IF
	END_IF
	
	// Lager 3 LT_Eingang
	IF Merler_L3_LTE = 0 THEN
	IF Flaschen[i_Zaehler].PY = -290 AND Flaschen[i_Zaehler].PX > 485 AND Flaschen[i_Zaehler].PX < 495
		THEN vis_Zuweisung.vis_i_Lager3_LT_Eingang := 0; Merler_L3_LTE := 1;
		ELSE vis_Zuweisung.vis_i_Lager3_LT_Eingang := 1;
	END_IF
	END_IF
	// Lager 2 LT_Eingang
	IF Merler_L2_LTE = 0 THEN
	IF Flaschen[i_Zaehler].PY = -390 AND Flaschen[i_Zaehler].PX > 485 AND Flaschen[i_Zaehler].PX < 495
		THEN vis_Zuweisung.vis_i_Lager2_LT_Eingang := 0; Merler_L2_LTE := 1;
		ELSE vis_Zuweisung.vis_i_Lager2_LT_Eingang := 1;
	END_IF
	END_IF
	
		// Lager 1 LT_Eingang
	IF Merler_L1_LTE = 0 THEN
	IF Flaschen[i_Zaehler].PX > 535 AND Flaschen[i_Zaehler].PX < 545 AND Flaschen[i_Zaehler].PY = -490
		THEN vis_Zuweisung.vis_i_Lager1_LT_Eingang := 0; Merler_L1_LTE := 1;
		ELSE vis_Zuweisung.vis_i_Lager1_LT_Eingang := 1;
	END_IF
	END_IF
	
	//Rücklauf LT_Ausgang
	IF Merker_RL_LTA = 0 THEN
	IF Flaschen[i_Zaehler].PY = -90 AND Flaschen[i_Zaehler].PX > 132 AND Flaschen[i_Zaehler].PX < 145
		THEN vis_Zuweisung.vis_i_Rueckl_LT_Ausgang := 0; Merker_RL_LTA := 1;
		ELSE vis_Zuweisung.vis_i_Rueckl_LT_Ausgang := 1; 
	END_IF
	END_IF
	
	// Lager 4 LT_Ausgang
	IF Merler_L4_LTA = 0 THEN
	IF Flaschen[i_Zaehler].PY = -190 AND Flaschen[i_Zaehler].PX > 132 AND Flaschen[i_Zaehler].PX < 145
		THEN vis_Zuweisung.vis_i_Lager4_LT_Ausgang := 0; Merler_L4_LTA := 1;
		ELSE vis_Zuweisung.vis_i_Lager4_LT_Ausgang := 1;
	END_IF
	END_IF
	
	// Lager 3 LT_Ausgang
	IF Merler_L3_LTA = 0 THEN
	IF Flaschen[i_Zaehler].PY = -290 AND Flaschen[i_Zaehler].PX > 132 AND Flaschen[i_Zaehler].PX < 145
		THEN vis_Zuweisung.vis_i_Lager3_LT_Ausgang := 0; Merler_L3_LTA := 1;
		ELSE vis_Zuweisung.vis_i_Lager3_LT_Ausgang := 1;
	END_IF
	END_IF
	
	// Lager 2 LT_Ausgang
	IF Merler_L2_LTA = 0 THEN
	IF Flaschen[i_Zaehler].PY = -390 AND Flaschen[i_Zaehler].PX > 132 AND Flaschen[i_Zaehler].PX < 145
		THEN vis_Zuweisung.vis_i_Lager2_LT_Ausgang := 0; Merler_L2_LTA := 1;
		ELSE vis_Zuweisung.vis_i_Lager2_LT_Ausgang := 1;
	END_IF
	END_IF
	
	// Lager 1 LT_Ausgang
	IF Merler_L1_LTA = 0 THEN 
	IF Flaschen[i_Zaehler].PY = -490 AND Flaschen[i_Zaehler].PX > 132 AND Flaschen[i_Zaehler].PX < 145
		THEN vis_Zuweisung.vis_i_Lager1_LT_Ausgang := 0; Merler_L1_LTA := 1;
		ELSE vis_Zuweisung.vis_i_Lager1_LT_Ausgang := 1;
	END_IF
	END_IF
	
END_FOR

IF vis_Zuweisung.vis_o_Sammelband_Richtung = 1 THEN vis_Zuweisung.Sammelband_RP := -90; ELSE vis_Zuweisung.Sammelband_RP := 90; END_IF

IF Anlageanaus = 0 THEN
	
	vis_Zuweisung.vis_i_Abtransport_LT		:= 0;
	vis_Zuweisung.vis_i_Annahme_LT_Eingang	:= 0;
	vis_Zuweisung.vis_i_Annahme_VE_heraus	:= 0;
	vis_Zuweisung.vis_i_Annahme_VE_hinein	:= 0;
	vis_Zuweisung.vis_i_Auto				:= 0;
	vis_Zuweisung.vis_i_BEKenn_LS_mitte		:= 0;
	vis_Zuweisung.vis_i_BEKenn_LS_oben		:= 0;
	vis_Zuweisung.vis_i_BEKenn_LS_unten		:= 0;
	vis_Zuweisung.vis_i_Lager1_LT_Ausgang	:= 0;
	vis_Zuweisung.vis_i_Lager1_LT_Eingang	:= 0;
	vis_Zuweisung.vis_i_Lager1_VE_heraus	:= 0;
	vis_Zuweisung.vis_i_Lager1_VE_hinein	:= 0;
	vis_Zuweisung.vis_i_Lager2_LT_Ausgang	:= 0;
	vis_Zuweisung.vis_i_Lager2_LT_Eingang	:= 0;
	vis_Zuweisung.vis_i_Lager2_VE_heraus	:= 0;
	vis_Zuweisung.vis_i_Lager2_VE_hinein	:= 0;
	vis_Zuweisung.vis_i_Lager2_We_gerade	:= 0;
	vis_Zuweisung.vis_i_Lager2_We_kurve		:= 0;
	vis_Zuweisung.vis_i_Lager3_LT_Ausgang	:= 0;
	vis_Zuweisung.vis_i_Lager3_LT_Eingang	:= 0;
	vis_Zuweisung.vis_i_Lager3_VE_heraus	:= 0;
	vis_Zuweisung.vis_i_Lager3_VE_hinein	:= 0;
	vis_Zuweisung.vis_i_Lager3_We_gerade	:= 0;
	vis_Zuweisung.vis_i_Lager3_We_kurve		:= 0;
	vis_Zuweisung.vis_i_Lager4_LT_Ausgang	:= 0;
	vis_Zuweisung.vis_i_Lager4_LT_Eingang	:= 0;
	vis_Zuweisung.vis_i_Lager4_VE_heraus	:= 0;
	vis_Zuweisung.vis_i_Lager4_VE_hinein	:= 0;
	vis_Zuweisung.vis_i_Lager4_We_gerade	:= 0;
	vis_Zuweisung.vis_i_Lager4_We_kurve		:= 0;
	vis_Zuweisung.vis_i_Rueckl_LT_Ausgang	:= 0;
	vis_Zuweisung.vis_i_Rueckl_LT_Eingang	:= 0;
	vis_Zuweisung.vis_i_Rueckl_VE_heraus	:= 0;
	vis_Zuweisung.vis_i_Rueckl_VE_hinein	:= 0;
	vis_Zuweisung.vis_i_Rueckl_We_gerade	:= 0;
	vis_Zuweisung.vis_i_Rueckl_We_kurve		:= 0;
	vis_Zuweisung.vis_i_Schritt				:= 0;
	vis_Zuweisung.vis_i_Weiter				:= 0;

END_IF




IF Anlageanaus = 0 OR vis_Zuweisung.vis_i_Notaus = 0 THEN
	
	vis_Zuweisung.vis_o_Annahme_Band		:= 0;
	//vis_Zuweisung.vis_o_Annahme_VE			:= 0;
	//vis_Zuweisung.vis_o_Lager1_Band			:= 0;
	//vis_Zuweisung.vis_o_Lager1_VE			:= 0;
	vis_Zuweisung.vis_o_Lager2_Band			:= 0;
	//vis_Zuweisung.vis_o_Lager2_VE			:= 0;
	//vis_Zuweisung.vis_o_Lager2_Weiche		:= 0;
	vis_Zuweisung.vis_o_Lager3_Band			:= 0;
	//vis_Zuweisung.vis_o_Lager3_VE			:= 0;
	//vis_Zuweisung.vis_o_Lager3_Weiche		:= 0;
	vis_Zuweisung.vis_o_Lager4_Band			:= 0;
	//vis_Zuweisung.vis_o_Lager4_VE			:= 0;
	//vis_Zuweisung.vis_o_Lager4_Weiche		:= 0;
	vis_Zuweisung.vis_o_Rueckl_Band			:= 0;
	//vis_Zuweisung.vis_o_Rueckl_VE			:= 0;
	//vis_Zuweisung.vis_o_Rueckl_Weiche		:= 0;
	vis_Zuweisung.vis_o_Sammelband_anaus	:= 0;
	vis_Zuweisung.vis_o_Sammelband_Richtung	:= 0;
	vis_Zuweisung.vis_o_Weichenband			:= 0;
	
END_IF

IF Anlageanaus = 0 THEN
	vis_Zuweisung.vis_o_Auto				:= 0;
	vis_Zuweisung.vis_o_Fehler				:= 0;
	vis_Zuweisung.vis_o_Schritt				:= 0;
	vis_Zuweisung.vis_o_Status				:= 0;
END_IF


// A5 Checkboxmanagement
A5_CB_FF(Clk:= Merker_A5_CB);
A5_CB_RF(CLK:=Merker_A5_CB);
IF A5_CB_FF.Q = TRUE THEN
FOR i_Zaehler := 1 TO 50 DO
	Flaschen[i_Zaehler].Aktiv := 0;
	Flaschen[i_Zaehler].PX := 0; 
	Flaschen[i_Zaehler].PY := 0 ;
	
END_FOR
END_IF
IF A5_CB_RF.Q = TRUE THEN
	FOR i_Zaehler := 1 TO 50 DO
	Flaschen[i_Zaehler].PX := Flaschen[i_Zaehler].PX  +300;
END_FOR
END_IF

END_PROGRAM

// vis_Zuweisung
PROGRAM vis_Zuweisung
VAR_INPUT
	(* Visualisierung Variabeln *)
	
	Sammelband_RP		:INT;
	Annahmeband_RP		:INT;
	Lager1_RP			:INT;
	Lager2_RP			:INT;
	Lager3_RP			:INT;
	Lager4_RP			:INT;
	Rueckl_RP			:INT;
	Weichenband_RP		:INT;
	Lager1_VE_rot		:INT;
	Lager2_VE_rot		:INT;
	Lager3_VE_rot		:INT;
	Lager4_VE_rot		:INT;
	Rueckl_VE_rot		:INT;
	Annahme_VE_rot		:INT;
	Lager1_Weiche_rot	:INT;
	Lager2_Weiche_rot	:INT;
	Lager3_Weiche_rot	:INT;
	Lager4_Weiche_rot	:INT;
	Rueckl_Weiche_rot	:INT;
	
	vis_i_Abtransport_LT		:BOOL;
	vis_i_Annahme_LT_Eingang	:BOOL;
	vis_i_Annahme_VE_heraus		:BOOL;
	vis_i_Annahme_VE_hinein		:BOOL;
	vis_i_Auto					:BOOL;
	vis_i_BEKenn_LS_mitte		:BOOL;
	vis_i_BEKenn_LS_oben		:BOOL;
	vis_i_BEKenn_LS_unten		:BOOL;
	vis_i_Lager1_LT_Ausgang		:BOOL;
	vis_i_Lager1_LT_Eingang		:BOOL;
	vis_i_Lager1_VE_heraus		:BOOL;
	vis_i_Lager1_VE_hinein		:BOOL;
	vis_i_Lager2_LT_Ausgang		:BOOL;
	vis_i_Lager2_LT_Eingang		:BOOL;
	vis_i_Lager2_VE_heraus		:BOOL;
	vis_i_Lager2_VE_hinein		:BOOL;
	vis_i_Lager2_We_gerade		:BOOL;
	vis_i_Lager2_We_kurve		:BOOL;
	vis_i_Lager3_LT_Ausgang		:BOOL;
	vis_i_Lager3_LT_Eingang		:BOOL;
	vis_i_Lager3_VE_heraus		:BOOL;
	vis_i_Lager3_VE_hinein		:BOOL;
	vis_i_Lager3_We_gerade		:BOOL;
	vis_i_Lager3_We_kurve		:BOOL;
	vis_i_Lager4_LT_Ausgang		:BOOL;
	vis_i_Lager4_LT_Eingang		:BOOL;
	vis_i_Lager4_VE_heraus		:BOOL;
	vis_i_Lager4_VE_hinein		:BOOL;
	vis_i_Lager4_We_gerade		:BOOL;
	vis_i_Lager4_We_kurve		:BOOL;
	vis_i_Notaus				:BOOL;
	vis_i_Quit					:BOOL;
	vis_i_Rueckl_LT_Ausgang		:BOOL;
	vis_i_Rueckl_LT_Eingang		:BOOL;
	vis_i_Rueckl_VE_heraus		:BOOL;
	vis_i_Rueckl_VE_hinein		:BOOL;
	vis_i_Rueckl_We_gerade		:BOOL;
	vis_i_Rueckl_We_kurve		:BOOL;
	vis_i_Schritt				:BOOL;
	vis_i_Weiter				:BOOL;
	
	
	vis_o_Annahme_Band			:BOOL;
	vis_o_Annahme_VE			:BOOL;
	vis_o_Auto					:BOOL;
	vis_o_Fehler				:BOOL;
	vis_o_Lager1_Band			:BOOL;
	vis_o_Lager1_VE				:BOOL;
	vis_o_Lager2_Band			:BOOL;
	vis_o_Lager2_VE				:BOOL;
	vis_o_Lager2_Weiche			:BOOL;
	vis_o_Lager3_Band			:BOOL;
	vis_o_Lager3_VE				:BOOL;
	vis_o_Lager3_Weiche			:BOOL;
	vis_o_Lager4_Band			:BOOL;
	vis_o_Lager4_VE				:BOOL;
	vis_o_Lager4_Weiche			:BOOL;
	vis_o_Rueckl_Band			:BOOL;
	vis_o_Rueckl_VE				:BOOL;
	vis_o_Rueckl_Weiche			:BOOL;
	vis_o_Sammelband_anaus		:BOOL;
	vis_o_Sammelband_Richtung	:BOOL;
	vis_o_Schritt				:BOOL;
	vis_o_Status				:BOOL;
	vis_o_Weichenband			:BOOL;
			
END_VAR

	IF vis_Ablauf.Anlageanaus = 1 AND vis_i_Notaus = 1   THEN
	(*Inputs*)
	GVL.i_Abtransport_LT		:= vis_i_Abtransport_LT;
	GVL.i_Annahme_LT_Eingang	:= vis_i_Annahme_LT_Eingang;
	GVL.i_Annahme_VE_heraus		:= vis_i_Annahme_VE_heraus	;
	GVL.i_Annahme_VE_hinein		:= vis_i_Annahme_VE_hinein	;
	GVL.i_Auto					:= vis_i_Auto;
	GVL.i_BEKenn_LS_mitte		:= vis_i_BEKenn_LS_mitte;
	GVL.i_BEKenn_LS_oben		:= vis_i_BEKenn_LS_oben;
	GVL.i_BEKenn_LT_unten		:= vis_i_BEKenn_LS_unten;
	GVL.i_Lager1_LT_Ausgang		:= vis_i_Lager1_LT_Ausgang;
	GVL.i_Lager1_LT_Eingang		:= vis_i_Lager1_LT_Eingang;
	GVL.i_Lager1_VE_heraus		:= vis_i_Lager1_VE_heraus;
	GVL.i_Lager1_VE_hinein		:= vis_i_Lager1_VE_hinein;
	GVL.i_Lager2_LT_Ausgang		:= vis_i_Lager2_LT_Ausgang;
	GVL.i_Lager2_LT_Eingang		:= vis_i_Lager2_LT_Eingang;
	GVL.i_Lager2_VE_heraus		:= vis_i_Lager2_VE_heraus;
	GVL.i_Lager2_VE_hinein		:= vis_i_Lager2_VE_hinein;
	GVL.i_Lager2_We_gerade		:= vis_i_Lager2_We_gerade;
	GVL.i_Lager2_We_kurve		:= vis_i_Lager2_We_kurve;
	GVL.i_Lager3_LT_Ausgang		:= vis_i_Lager3_LT_Ausgang;
	GVL.i_Lager3_LT_Eingang		:= vis_i_Lager3_LT_Eingang	;
	GVL.i_Lager3_VE_heraus		:= vis_i_Lager3_VE_heraus;
	GVL.i_Lager3_VE_hinein		:= vis_i_Lager3_VE_hinein;
	GVL.i_Lager3_We_gerade		:= vis_i_Lager3_We_gerade;
	GVL.i_Lager3_We_kurve		:= vis_i_Lager3_We_kurve;
	GVL.i_Lager4_LT_Ausgang		:= vis_i_Lager4_LT_Ausgang;
	GVL.i_Lager4_LT_Eingang		:= vis_i_Lager4_LT_Eingang;
	GVL.i_Lager4_VE_heraus		:= vis_i_Lager4_VE_heraus;
	GVL.i_Lager4_VE_hinein		:= vis_i_Lager4_VE_hinein;
	GVL.i_Lager4_We_gerade		:= vis_i_Lager4_We_gerade;
	GVL.i_Lager4_We_kurve		:= vis_i_Lager4_We_kurve;
	GVL.i_Notaus				:= vis_i_Notaus;
	GVL.i_Quit					:= vis_i_Quit;
	GVL.i_Rueckl_LT_Ausgang		:= vis_i_Rueckl_LT_Ausgang;
	GVL.i_Rueckl_LT_Eingang		:= vis_i_Rueckl_LT_Eingang;
	GVL.i_Rueckl_VE_heraus		:= vis_i_Rueckl_VE_heraus;
	GVL.i_Rueckl_VE_hinein		:= vis_i_Rueckl_VE_hinein;
	GVL.i_Rueckl_We_gerade		:= vis_i_Rueckl_We_gerade;
	GVL.i_Rueckl_We_kurve		:= vis_i_Rueckl_We_kurve	;
	GVL.i_Schritt				:= vis_i_Schritt;
	GVL.i_Weiter				:= vis_i_Weiter;
	
	(*Outputs*)
	vis_o_Annahme_VE			:= GVL.o_Annahme_VE;
	vis_o_Auto					:= GVL.o_Auto;
	vis_o_Fehler				:= GVL.o_Fehler;
	vis_o_Lager1_VE				:= GVL.o_Lager1_VE;
	vis_o_Lager2_VE				:= GVL.o_Lager2_VE;
	vis_o_Lager2_Weiche			:= GVL.o_Lager2_Weiche;
	vis_o_Lager3_VE				:= GVL.o_Lager3_VE;
	vis_o_Lager3_Weiche			:= GVL.o_Lager3_Weiche;
	vis_o_Lager4_VE				:= GVL.o_Lager4_VE;
	vis_o_Lager4_Weiche			:= GVL.o_Lager4_Weiche;
	vis_o_Rueckl_VE				:= GVL.o_Rueckl_VE;
	vis_o_Rueckl_Weiche			:= GVL.o_Rueckl_Weiche;
	vis_o_Sammelband_Richtung	:= GVL.o_Sammelband_Richtung;
	vis_o_Schritt				:= GVL.o_Schritt;
	vis_o_Status				:= GVL.o_Status;
	vis_o_Weichenband			:= GVL.o_Weichenband;
	vis_o_Rueckl_Band			:= GVL.o_Rueckl_Band;
	vis_o_Annahme_Band			:= GVL.o_Annahme_Band;
	vis_o_Lager1_Band			:= GVL.o_Lager1_Band;	
	vis_o_Lager2_Band			:= GVL.o_Lager2_Band;
	vis_o_Lager3_Band			:= GVL.o_Lager3_Band;
	vis_o_Lager4_Band			:= GVL.o_Lager4_Band;
	vis_o_Sammelband_anaus		:= GVL.o_Sammelband_anaus;
	ELSIF vis_Zuweisung.vis_i_Notaus = FALSE AND vis_Ablauf.Anlageanaus = TRUE THEN
	(*Inputs*)
	GVL.i_Abtransport_LT		:= vis_i_Abtransport_LT;
	GVL.i_Annahme_LT_Eingang	:= vis_i_Annahme_LT_Eingang;
	GVL.i_Annahme_VE_heraus		:= vis_i_Annahme_VE_heraus	;
	GVL.i_Annahme_VE_hinein		:= vis_i_Annahme_VE_hinein	;
	GVL.i_Auto					:= vis_i_Auto;
	GVL.i_BEKenn_LS_mitte		:= vis_i_BEKenn_LS_mitte;
	GVL.i_BEKenn_LS_oben		:= vis_i_BEKenn_LS_oben;
	GVL.i_BEKenn_LT_unten		:= vis_i_BEKenn_LS_unten;
	GVL.i_Lager1_LT_Ausgang		:= vis_i_Lager1_LT_Ausgang;
	GVL.i_Lager1_LT_Eingang		:= vis_i_Lager1_LT_Eingang;
	GVL.i_Lager1_VE_heraus		:= vis_i_Lager1_VE_heraus;
	GVL.i_Lager1_VE_hinein		:= vis_i_Lager1_VE_hinein;
	GVL.i_Lager2_LT_Ausgang		:= vis_i_Lager2_LT_Ausgang;
	GVL.i_Lager2_LT_Eingang		:= vis_i_Lager2_LT_Eingang;
	GVL.i_Lager2_VE_heraus		:= vis_i_Lager2_VE_heraus;
	GVL.i_Lager2_VE_hinein		:= vis_i_Lager2_VE_hinein;
	GVL.i_Lager2_We_gerade		:= vis_i_Lager2_We_gerade;
	GVL.i_Lager2_We_kurve		:= vis_i_Lager2_We_kurve;
	GVL.i_Lager3_LT_Ausgang		:= vis_i_Lager3_LT_Ausgang;
	GVL.i_Lager3_LT_Eingang		:= vis_i_Lager3_LT_Eingang	;
	GVL.i_Lager3_VE_heraus		:= vis_i_Lager3_VE_heraus;
	GVL.i_Lager3_VE_hinein		:= vis_i_Lager3_VE_hinein;
	GVL.i_Lager3_We_gerade		:= vis_i_Lager3_We_gerade;
	GVL.i_Lager3_We_kurve		:= vis_i_Lager3_We_kurve;
	GVL.i_Lager4_LT_Ausgang		:= vis_i_Lager4_LT_Ausgang;
	GVL.i_Lager4_LT_Eingang		:= vis_i_Lager4_LT_Eingang;
	GVL.i_Lager4_VE_heraus		:= vis_i_Lager4_VE_heraus;
	GVL.i_Lager4_VE_hinein		:= vis_i_Lager4_VE_hinein;
	GVL.i_Lager4_We_gerade		:= vis_i_Lager4_We_gerade;
	GVL.i_Lager4_We_kurve		:= vis_i_Lager4_We_kurve;
	GVL.i_Notaus				:= vis_i_Notaus;
	GVL.i_Quit					:= vis_i_Quit;
	GVL.i_Rueckl_LT_Ausgang		:= vis_i_Rueckl_LT_Ausgang;
	GVL.i_Rueckl_LT_Eingang		:= vis_i_Rueckl_LT_Eingang;
	GVL.i_Rueckl_VE_heraus		:= vis_i_Rueckl_VE_heraus;
	GVL.i_Rueckl_VE_hinein		:= vis_i_Rueckl_VE_hinein;
	GVL.i_Rueckl_We_gerade		:= vis_i_Rueckl_We_gerade;
	GVL.i_Rueckl_We_kurve		:= vis_i_Rueckl_We_kurve	;
	GVL.i_Schritt				:= vis_i_Schritt;
	GVL.i_Weiter				:= vis_i_Weiter;
	
	(*Outputs*)
	vis_o_Annahme_VE			:= GVL.o_Annahme_VE;
	vis_o_Auto					:= GVL.o_Auto;
	vis_o_Fehler				:= GVL.o_Fehler;
	vis_o_Lager1_VE				:= GVL.o_Lager1_VE;
	vis_o_Lager2_VE				:= GVL.o_Lager2_VE;
	vis_o_Lager2_Weiche			:= GVL.o_Lager2_Weiche;
	vis_o_Lager3_VE				:= GVL.o_Lager3_VE;
	vis_o_Lager3_Weiche			:= GVL.o_Lager3_Weiche;
	vis_o_Lager4_VE				:= GVL.o_Lager4_VE;
	vis_o_Lager4_Weiche			:= GVL.o_Lager4_Weiche;
	vis_o_Rueckl_VE				:= GVL.o_Rueckl_VE;
	vis_o_Rueckl_Weiche			:= GVL.o_Rueckl_Weiche;
	vis_o_Sammelband_Richtung	:= GVL.o_Sammelband_Richtung;
	vis_o_Schritt				:= GVL.o_Schritt;
	vis_o_Status				:= GVL.o_Status;
	vis_o_Weichenband			:= 0;
	vis_o_Rueckl_Band			:= 0;
	vis_o_Annahme_Band			:= 0;
	vis_o_Lager1_Band			:= 0;	
	vis_o_Lager2_Band			:= 0;
	vis_o_Lager3_Band			:= 0;
	vis_o_Lager4_Band			:= 0;
	vis_o_Sammelband_anaus		:= 0;
	END_IF

END_PROGRAM

// SoftSPS/Application/Visualization
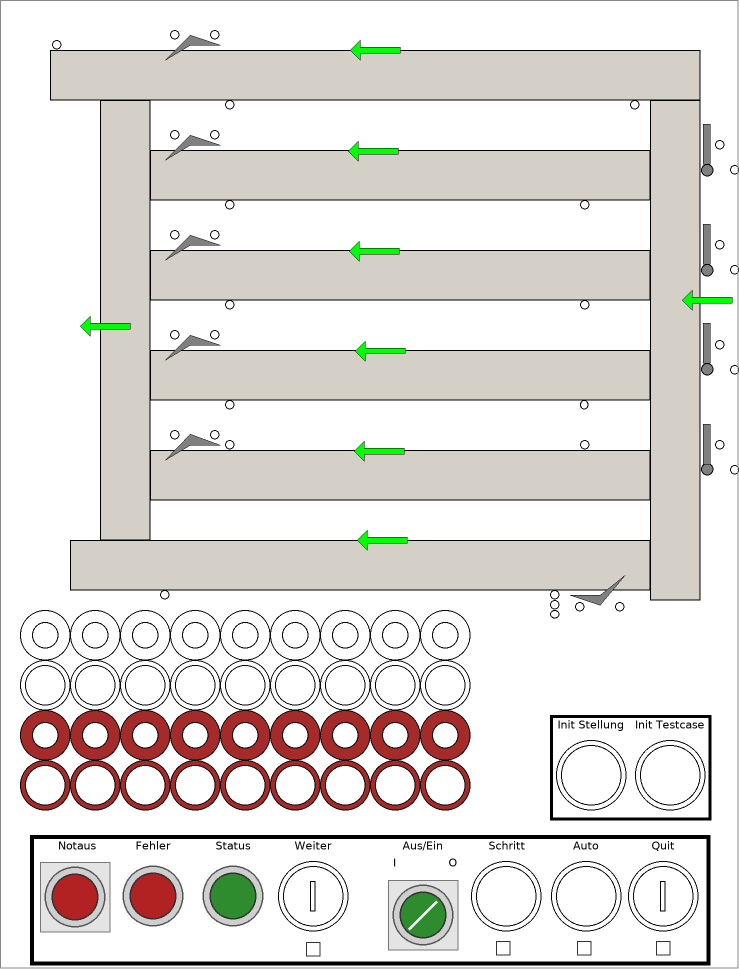
VISUALIZATION Visualization  // 739x969
    Rectangle (30,835 680x130)
    Rectangle (50,50 650x50)
    Rectangle (100,100 50x440)
    Rectangle (150,150 500x50)
    Rectangle (150,250 500x50)
    Rectangle (150,350 500x50)
    Rectangle (150,450 500x50)
    Rectangle (70,540 580x50)
    Rectangle (650,100 50x500)
    Ellipse (225,100 9x9), tooltip "i_Lager1_LT_Ausgang", colour toggle: vis_Zuweisung.vis_i_Lager1_LT_Ausgang
    Ellipse (225,200 9x9), tooltip "i_Lager2_LT_Ausgang", colour toggle: vis_Zuweisung.vis_i_Lager2_LT_Ausgang
    Ellipse (225,300 9x9), tooltip "i_Lager3_LT_Ausgang", colour toggle: vis_Zuweisung.vis_i_Lager3_LT_Ausgang
    Ellipse (225,400 9x9), tooltip "i_Lager4_LT_Ausgang", colour toggle: vis_Zuweisung.vis_i_Lager4_LT_Ausgang
    Ellipse (225,440 9x9), tooltip "i_Rueckl_LT_Ausgang", colour toggle: vis_Zuweisung.vis_i_Rueckl_LT_Ausgang
    Ellipse (160,590 9x9), tooltip "i_Annahme_LT_Eingang", colour toggle: vis_Zuweisung.vis_i_Annahme_LT_Eingang
    Ellipse (550,590 9x9), tooltip "i_BEKenn_LS_oben", colour toggle: vis_Zuweisung.vis_i_BEKenn_LS_oben
    Ellipse (550,600 9x9), tooltip "i_BEKenn_LS_mitte", colour toggle: vis_Zuweisung.vis_i_BEKenn_LS_mitte
    Ellipse (550,610 9x8), tooltip "i_BEKenn_LT_unten", colour toggle: vis_Zuweisung.vis_i_BEKenn_LS_unten
    Ellipse (580,440 9x9), tooltip "i_Rueckl_LT_Eingang", colour toggle: vis_Zuweisung.vis_i_Rueckl_LT_Eingang
    Ellipse (580,400 8x9), tooltip "i_Lager4_LT_Eingang", colour toggle: vis_Zuweisung.vis_i_Lager4_LT_Eingang
    Ellipse (580,300 9x9), tooltip "i_Lager3_LT_Eingang", colour toggle: vis_Zuweisung.vis_i_Lager3_LT_Eingang
    Ellipse (580,200 9x9), tooltip "i_Lager2_LT_Eingang", colour toggle: vis_Zuweisung.vis_i_Lager2_LT_Eingang
    Ellipse (630,100 9x9), tooltip "i_Lager1_LT_Eingang", colour toggle: vis_Zuweisung.vis_i_Lager1_LT_Eingang
    Polygon (190,445) (165,460) (190,434) (220,445)
        p2858320360: vis_Zuweisung.Rueckl_VE_rot
    Polygon (190,345) (165,360) (190,335) (220,345)
        p2858320360: vis_Zuweisung.Lager4_VE_rot
    Polygon (190,245) (165,260) (190,235) (220,245)
        p2858320360: vis_Zuweisung.Lager3_VE_rot
    Polygon (190,145) (165,160) (190,135) (220,145)
        p2858320360: vis_Zuweisung.Lager2_VE_rot
    Polygon (190,45) (165,60) (190,35) (220,45)
        p2858320360: vis_Zuweisung.Lager1_VE_rot
    Polygon (600,605) (570,595) (600,595) (625,575)
        p2858320360: vis_Zuweisung.Annahme_VE_rot
    Polygon (399,254) (359,254) (359,261) (349,251) (359,241) (359,248) (399,248), invisible if: vis_Zuweisung.vis_o_Lager3_Band = 0
        p2858320360: vis_Zuweisung.Lager3_RP
    Polygon (405,353) (365,353) (365,361) (355,351) (365,341) (365,348) (405,348), invisible if: vis_Zuweisung.vis_o_Lager4_Band = 0
        p2858320360: vis_Zuweisung.Lager4_RP
    Polygon (404,454) (364,454) (364,461) (354,451) (364,441) (364,448) (404,448), invisible if: vis_Zuweisung.vis_o_Rueckl_Band = 0
        p2858320360: vis_Zuweisung.Rueckl_RP
    Polygon (398,154) (358,154) (358,161) (348,151) (358,141) (358,148) (398,148), invisible if: vis_Zuweisung.vis_o_Lager2_Band = 0
        p2858320360: vis_Zuweisung.Lager2_RP
    Polygon (400,53) (360,53) (360,60) (350,50) (360,40) (360,47) (400,47), invisible if: vis_Zuweisung.vis_o_Lager1_Band = 0
        p2858320360: vis_Zuweisung.Lager1_RP
    Polygon (407,543) (367,543) (367,550) (357,540) (367,530) (367,537) (407,537), invisible if: vis_Zuweisung.vis_o_Annahme_Band = 0
    Polygon (130,329) (90,329) (90,336) (80,326) (90,316) (90,323) (130,323), invisible if: vis_Zuweisung.vis_o_Sammelband_anaus = 0
        p2858320360: vis_Zuweisung.Sammelband_RP
    Polygon (732,303) (692,303) (692,310) (682,300) (692,290) (692,297) (732,297), invisible if: vis_Zuweisung.vis_o_Weichenband = 0
    Ellipse (701,164 12x12)
    Ellipse (701,264 12x12)
    Ellipse (701,363 12x12)
    Ellipse (701,463 12x12)
    Group (20,610 50x50)
        p2738717112: (vis_Ablauf.Flaschen[1].PY -70)*vis_Ablauf.Flaschen[1].Aktiv
        p3560616238: (vis_Ablauf.Flaschen[1].PX +50)*vis_Ablauf.Flaschen[1].Aktiv
        tap vis_Ablauf.Taster_Flasche[1]
        Ellipse (0,0 50x50)
        Ellipse (12,12 26x26)
    Group (70,610 50x50)
        p3560616238: (vis_Ablauf.Flaschen[2].PX)*vis_Ablauf.Flaschen[2].Aktiv
        p2738717112: (vis_Ablauf.Flaschen[2].PY -70)*vis_Ablauf.Flaschen[2].Aktiv
        tap vis_Ablauf.Taster_Flasche[2]
        Ellipse (0,0 50x50)
        Ellipse (12,12 26x26)
    Group (120,610 50x50)
        p3560616238: (vis_Ablauf.Flaschen[3].PX -50)*vis_Ablauf.Flaschen[3].Aktiv
        p2738717112: (vis_Ablauf.Flaschen[3].PY -70)*vis_Ablauf.Flaschen[3].Aktiv
        tap vis_Ablauf.Taster_Flasche[3]
        Ellipse (0,0 50x50)
        Ellipse (12,12 26x26)
    Group (220,610 50x50)
        p3560616238: (vis_Ablauf.Flaschen[5].PX -150)*vis_Ablauf.Flaschen[5].Aktiv
        p2738717112: (vis_Ablauf.Flaschen[5].PY -70)*vis_Ablauf.Flaschen[5].Aktiv
        tap vis_Ablauf.Taster_Flasche[5]
        Ellipse (0,0 50x50)
        Ellipse (12,12 26x26)
    Group (170,610 50x50)
        p3560616238: (vis_Ablauf.Flaschen[4].PX -100)*vis_Ablauf.Flaschen[4].Aktiv
        p2738717112: (vis_Ablauf.Flaschen[4].PY -70)*vis_Ablauf.Flaschen[4].Aktiv
        tap vis_Ablauf.Taster_Flasche[4]
        Ellipse (0,0 50x50)
        Ellipse (12,12 26x26)
    Polygon (703,464) (703,424) (710,424) (710,464)
        p2858320360: vis_Zuweisung.Rueckl_Weiche_rot
    Polygon (703,363) (703,323) (710,323) (710,363)
        p2858320360: vis_Zuweisung.Lager4_Weiche_rot
    Polygon (703,264) (703,224) (710,224) (710,264)
        p2858320360: vis_Zuweisung.Lager3_Weiche_rot
    Polygon (703,164) (703,124) (710,124) (710,164)
        p2858320360: vis_Zuweisung.Lager2_Weiche_rot
    RotarySwitch (388,861 70x108), variable: vis_Ablauf.Anlageanaus, style: Switch-RotarySwitch-Green
    PushSwitchLed (40,862 70x70), variable: vis_Zuweisung.vis_i_Notaus, behaviour: TOGGLE, style: Switch-PushSwitchLed-Red
    Lamp1 (118,861 70x70), variable: vis_Zuweisung.vis_o_Fehler, style: Lamp-Lamp1-Red
    Lamp1 (198,861 70x70), variable: vis_Zuweisung.vis_o_Status, style: Lamp-Lamp1-Green
    Ellipse (278,861 70x70)
    Ellipse (628,861 70x70)
    Group (283,866 60x60)
        tap vis_Zuweisung.vis_i_Weiter
        Ellipse (0,0 60x60)
        RoundedRectangle (27,15 5x30)
    Group (633,866 60x60)
        tap vis_Zuweisung.vis_i_Quit
        Ellipse (0,0 60x60)
        RoundedRectangle (27,15 5x30)
    Label (628,831 70x30), "Quit"
    Label (551,831 70x30), "Auto"
    Label (472,831 70x30), "Schritt"
    Label (388,831 70x30), "Aus/Ein"
    Label (278,831 70x30), "Weiter"
    Label (198,831 70x30), "Status"
    Label (118,831 70x30), "Fehler"
    Label (42,831 70x30), "Notaus"
    Group (270,610 50x50)
        p3560616238: (vis_Ablauf.Flaschen[6].PX -200)*vis_Ablauf.Flaschen[6].Aktiv
        p2738717112: (vis_Ablauf.Flaschen[6].PY -70)*vis_Ablauf.Flaschen[6].Aktiv
        tap vis_Ablauf.Taster_Flasche[6]
        Ellipse (0,0 50x50)
        Ellipse (12,12 26x26)
    Group (320,610 50x50)
        p3560616238: (vis_Ablauf.Flaschen[7].PX -250)*vis_Ablauf.Flaschen[7].Aktiv
        p2738717112: (vis_Ablauf.Flaschen[7].PY -70)*vis_Ablauf.Flaschen[7].Aktiv
        tap vis_Ablauf.Taster_Flasche[7]
        Ellipse (0,0 50x50)
        Ellipse (12,12 26x26)
    Group (20,760 50x50)
        p3560616238: (vis_Ablauf.Flaschen[30].PX +50)*vis_Ablauf.Flaschen[30].Aktiv
        p2738717112: (vis_Ablauf.Flaschen[30].PY -220)*vis_Ablauf.Flaschen[30].Aktiv
        tap vis_Ablauf.Taster_Flasche[30]
        Ellipse (0,0 50x50)
        Ellipse (5,5 40x40)
    Group (20,660 50x50)
        p3560616238: (vis_Ablauf.Flaschen[10].PX +50)*vis_Ablauf.Flaschen[10].Aktiv
        p2738717112: (vis_Ablauf.Flaschen[10].PY -120)*vis_Ablauf.Flaschen[10].Aktiv
        tap vis_Ablauf.Taster_Flasche[10]
        Ellipse (0,0 50x50)
        Ellipse (5,5 40x40)
    Group (70,660 50x50)
        p3560616238: (vis_Ablauf.Flaschen[11].PX)*vis_Ablauf.Flaschen[11].Aktiv
        p2738717112: (vis_Ablauf.Flaschen[11].PY -120)*vis_Ablauf.Flaschen[11].Aktiv
        tap vis_Ablauf.Taster_Flasche[11]
        Ellipse (0,0 50x50)
        Ellipse (5,5 40x40)
    Group (120,660 50x50)
        p3560616238: (vis_Ablauf.Flaschen[12].PX -50)*vis_Ablauf.Flaschen[12].Aktiv
        p2738717112: (vis_Ablauf.Flaschen[12].PY -120)*vis_Ablauf.Flaschen[12].Aktiv
        tap vis_Ablauf.Taster_Flasche[12]
        Ellipse (0,0 50x50)
        Ellipse (5,5 40x40)
    Group (170,660 50x50)
        p3560616238: (vis_Ablauf.Flaschen[13].PX -100)*vis_Ablauf.Flaschen[13].Aktiv
        p2738717112: (vis_Ablauf.Flaschen[13].PY -120)*vis_Ablauf.Flaschen[13].Aktiv
        tap vis_Ablauf.Taster_Flasche[13]
        Ellipse (0,0 50x50)
        Ellipse (5,5 40x40)
    Group (220,660 50x50)
        p3560616238: (vis_Ablauf.Flaschen[14].PX -150)*vis_Ablauf.Flaschen[14].Aktiv
        p2738717112: (vis_Ablauf.Flaschen[14].PY -120)*vis_Ablauf.Flaschen[14].Aktiv
        tap vis_Ablauf.Taster_Flasche[14]
        Ellipse (0,0 50x50)
        Ellipse (5,5 40x40)
    Group (270,660 50x50)
        p3560616238: (vis_Ablauf.Flaschen[15].PX -200)*vis_Ablauf.Flaschen[15].Aktiv
        p2738717112: (vis_Ablauf.Flaschen[15].PY -120)*vis_Ablauf.Flaschen[15].Aktiv
        tap vis_Ablauf.Taster_Flasche[15]
        Ellipse (0,0 50x50)
        Ellipse (5,5 40x40)
    Group (320,660 50x50)
        p3560616238: (vis_Ablauf.Flaschen[16].PX -250)*vis_Ablauf.Flaschen[16].Aktiv
        p2738717112: (vis_Ablauf.Flaschen[16].PY -120)*vis_Ablauf.Flaschen[16].Aktiv
        tap vis_Ablauf.Taster_Flasche[16]
        Ellipse (0,0 50x50)
        Ellipse (5,5 40x40)
    Group (20,710 50x50)
        p3560616238: (vis_Ablauf.Flaschen[20].PX +50)*vis_Ablauf.Flaschen[20].Aktiv
        p2738717112: (vis_Ablauf.Flaschen[20].PY -170)*vis_Ablauf.Flaschen[20].Aktiv
        tap vis_Ablauf.Taster_Flasche[20]
        Ellipse (0,0 50x50)
            tap vis_Ablauf.Taster_Flasche[20]
        Ellipse (12,12 26x26)
    Group (70,710 50x50)
        p3560616238: (vis_Ablauf.Flaschen[21].PX)*vis_Ablauf.Flaschen[21].Aktiv
        p2738717112: (vis_Ablauf.Flaschen[21].PY -170)*vis_Ablauf.Flaschen[21].Aktiv
        tap vis_Ablauf.Taster_Flasche[21]
        Ellipse (0,0 50x50)
            tap vis_Ablauf.Taster_Flasche[20]
        Ellipse (12,12 26x26)
    Group (120,710 50x50)
        p3560616238: (vis_Ablauf.Flaschen[22].PX -50)*vis_Ablauf.Flaschen[22].Aktiv
        p2738717112: (vis_Ablauf.Flaschen[22].PY -170)*vis_Ablauf.Flaschen[22].Aktiv
        tap vis_Ablauf.Taster_Flasche[22]
        Ellipse (0,0 50x50)
            tap vis_Ablauf.Taster_Flasche[20]
        Ellipse (12,12 26x26)
    Group (170,710 50x50)
        p3560616238: (vis_Ablauf.Flaschen[23].PX -100)*vis_Ablauf.Flaschen[23].Aktiv
        p2738717112: (vis_Ablauf.Flaschen[23].PY -170)*vis_Ablauf.Flaschen[23].Aktiv
        tap vis_Ablauf.Taster_Flasche[23]
        Ellipse (0,0 50x50)
            tap vis_Ablauf.Taster_Flasche[20]
        Ellipse (12,12 26x26)
    Group (220,710 50x50)
        p3560616238: (vis_Ablauf.Flaschen[24].PX -150)*vis_Ablauf.Flaschen[24].Aktiv
        p2738717112: (vis_Ablauf.Flaschen[24].PY -170)*vis_Ablauf.Flaschen[24].Aktiv
        tap vis_Ablauf.Taster_Flasche[24]
        Ellipse (0,0 50x50)
            tap vis_Ablauf.Taster_Flasche[20]
        Ellipse (12,12 26x26)
    Group (270,710 50x50)
        p3560616238: (vis_Ablauf.Flaschen[25].PX -200)*vis_Ablauf.Flaschen[25].Aktiv
        p2738717112: (vis_Ablauf.Flaschen[25].PY -170)*vis_Ablauf.Flaschen[25].Aktiv
        tap vis_Ablauf.Taster_Flasche[25]
        Ellipse (0,0 50x50)
            tap vis_Ablauf.Taster_Flasche[20]
        Ellipse (12,12 26x26)
    Group (320,710 50x50)
        p3560616238: (vis_Ablauf.Flaschen[26].PX -250)*vis_Ablauf.Flaschen[26].Aktiv
        p2738717112: (vis_Ablauf.Flaschen[26].PY -170)*vis_Ablauf.Flaschen[26].Aktiv
        tap vis_Ablauf.Taster_Flasche[26]
        Ellipse (0,0 50x50)
            tap vis_Ablauf.Taster_Flasche[20]
        Ellipse (12,12 26x26)
    Group (70,760 50x50)
        p3560616238: (vis_Ablauf.Flaschen[31].PX )*vis_Ablauf.Flaschen[31].Aktiv
        p2738717112: (vis_Ablauf.Flaschen[31].PY -220)*vis_Ablauf.Flaschen[31].Aktiv
        tap vis_Ablauf.Taster_Flasche[31]
        Ellipse (0,0 50x50)
        Ellipse (5,5 40x40)
    Group (120,760 50x50)
        p3560616238: (vis_Ablauf.Flaschen[32].PX - 50 )*vis_Ablauf.Flaschen[32].Aktiv
        p2738717112: (vis_Ablauf.Flaschen[32].PY -220)*vis_Ablauf.Flaschen[32].Aktiv
        tap vis_Ablauf.Taster_Flasche[32]
        Ellipse (0,0 50x50)
        Ellipse (5,5 40x40)
    Group (170,760 50x50)
        p3560616238: (vis_Ablauf.Flaschen[33].PX - 100 )*vis_Ablauf.Flaschen[33].Aktiv
        p2738717112: (vis_Ablauf.Flaschen[33].PY -220)*vis_Ablauf.Flaschen[33].Aktiv
        tap vis_Ablauf.Taster_Flasche[33]
        Ellipse (0,0 50x50)
        Ellipse (5,5 40x40)
    Group (220,760 50x50)
        p3560616238: (vis_Ablauf.Flaschen[34].PX - 150 )*vis_Ablauf.Flaschen[34].Aktiv
        p2738717112: (vis_Ablauf.Flaschen[34].PY -220)*vis_Ablauf.Flaschen[34].Aktiv
        tap vis_Ablauf.Taster_Flasche[34]
        Ellipse (0,0 50x50)
        Ellipse (5,5 40x40)
    Group (270,760 50x50)
        p3560616238: (vis_Ablauf.Flaschen[35].PX - 200 )*vis_Ablauf.Flaschen[35].Aktiv
        p2738717112: (vis_Ablauf.Flaschen[35].PY -220)*vis_Ablauf.Flaschen[35].Aktiv
        tap vis_Ablauf.Taster_Flasche[35]
        Ellipse (0,0 50x50)
        Ellipse (5,5 40x40)
    Group (320,760 50x50)
        p3560616238: (vis_Ablauf.Flaschen[36].PX - 250 )*vis_Ablauf.Flaschen[36].Aktiv
        p2738717112: (vis_Ablauf.Flaschen[36].PY -220)*vis_Ablauf.Flaschen[36].Aktiv
        tap vis_Ablauf.Taster_Flasche[36]
        Ellipse (0,0 50x50)
        Ellipse (5,5 40x40)
    Ellipse (210,330 9x9), tooltip "i_Lager4_VE_hinein", colour toggle: vis_Zuweisung.vis_i_Lager4_VE_hinein
    Ellipse (170,330 9x9), tooltip "i_Lager4_VE_heraus", colour toggle: vis_Zuweisung.vis_i_Lager4_VE_heraus
    Ellipse (210,430 9x9), tooltip "i_Rueckl_VE_hinein", colour toggle: vis_Zuweisung.vis_i_Rueckl_VE_hinein
    Ellipse (170,430 9x9), tooltip "i_Rueckl_VE_heraus", colour toggle: vis_Zuweisung.vis_i_Rueckl_VE_heraus
    Ellipse (210,230 9x9), tooltip "i_Lager3_VE_hinein", colour toggle: vis_Zuweisung.vis_i_Lager3_VE_hinein
    Ellipse (170,230 9x9), tooltip "i_Lager3_VE_heraus", colour toggle: vis_Zuweisung.vis_i_Lager3_VE_heraus
    Ellipse (210,130 9x9), tooltip "i_Lager2_VE_hinein", colour toggle: vis_Zuweisung.vis_i_Lager2_VE_hinein
    Ellipse (170,130 9x9), tooltip "i_Lager2_VE_heraus", colour toggle: vis_Zuweisung.vis_i_Lager2_VE_heraus
    Ellipse (210,30 9x9), tooltip "i_Lager1_VE_hinein", colour toggle: vis_Zuweisung.vis_i_Lager1_VE_hinein
    Ellipse (170,30 9x9), tooltip "i_Lager1_VE_heraus", colour toggle: vis_Zuweisung.vis_i_Lager1_VE_heraus
    Ellipse (615,602 9x9), tooltip "i_Annahme_VE_heraus", colour toggle: vis_Zuweisung.vis_i_Annahme_VE_heraus
    Ellipse (575,602 9x9), tooltip "i_Annahme_VE_hinein", colour toggle: vis_Zuweisung.vis_i_Annahme_VE_hinein
    Ellipse (730,465 9x9), tooltip "i_Rueckl_We_gerade", colour toggle: vis_Zuweisung.vis_i_Rueckl_We_gerade
    Ellipse (715,440 9x9), tooltip "i_Rueckl_We_kurve", colour toggle: vis_Zuweisung.vis_i_Rueckl_We_kurve
    Ellipse (730,365 9x9), tooltip "i_Lager4_We_gerade", colour toggle: vis_Zuweisung.vis_i_Lager4_We_gerade
    Ellipse (715,340 9x9), tooltip "i_Lager4_We_kurve", colour toggle: vis_Zuweisung.vis_i_Lager4_We_kurve
    Ellipse (730,265 9x9), tooltip "i_Lager3_We_gerade", colour toggle: vis_Zuweisung.vis_i_Lager3_We_gerade
    Ellipse (715,240 9x9), tooltip "i_Lager3_We_kurve", colour toggle: vis_Zuweisung.vis_i_Lager3_We_kurve
    Ellipse (730,165 9x9), tooltip "i_Lager2_We_gerade", colour toggle: vis_Zuweisung.vis_i_Lager2_We_gerade
    Ellipse (715,140 9x9), tooltip "i_Lager2_We_kurve", colour toggle: vis_Zuweisung.vis_i_Lager2_We_kurve
    Label (350,848 150x30), "I O"
    Checkbox (654,936 23x24), variable: vis_Zuweisung.vis_i_Quit
    Checkbox (575,936 26x24), variable: vis_Zuweisung.vis_i_Auto
    Checkbox (494,936 24x24), variable: vis_Zuweisung.vis_i_Schritt
    Checkbox (304,937 24x24), variable: vis_Zuweisung.vis_i_Weiter
    Ellipse (52,40 9x9), tooltip "i_Abtransport_LT", colour toggle: vis_Zuweisung.vis_i_Abtransport_LT
    Ellipse (551,861 70x70)
    Ellipse (471,861 70x70)
    Ellipse (556,866 60x60), colour toggle: vis_Zuweisung.vis_o_Auto
        tap vis_Zuweisung.vis_i_Auto
    Ellipse (476,866 60x60), colour toggle: vis_Zuweisung.vis_o_Schritt
        tap vis_Zuweisung.vis_i_Schritt
    Group (370,610 50x50)
        p3560616238: (vis_Ablauf.Flaschen[8].PX -300)*vis_Ablauf.Flaschen[8].Aktiv
        p2738717112: (vis_Ablauf.Flaschen[8].PY -70)*vis_Ablauf.Flaschen[8].Aktiv
        tap vis_Ablauf.Taster_Flasche[8]
        Ellipse (0,0 50x50)
        Ellipse (12,12 26x26)
    Group (420,610 50x50)
        p3560616238: (vis_Ablauf.Flaschen[9].PX -350)*vis_Ablauf.Flaschen[9].Aktiv
        p2738717112: (vis_Ablauf.Flaschen[9].PY -70)*vis_Ablauf.Flaschen[9].Aktiv
        tap vis_Ablauf.Taster_Flasche[9]
        Ellipse (0,0 50x50)
        Ellipse (12,12 26x26)
    Group (420,660 50x50)
        p3560616238: (vis_Ablauf.Flaschen[18].PX -350)*vis_Ablauf.Flaschen[18].Aktiv
        p2738717112: (vis_Ablauf.Flaschen[18].PY -120)*vis_Ablauf.Flaschen[18].Aktiv
        tap vis_Ablauf.Taster_Flasche[18]
        Ellipse (0,0 50x50)
        Ellipse (5,5 40x40)
    Group (370,660 50x50)
        p3560616238: (vis_Ablauf.Flaschen[17].PX -300)*vis_Ablauf.Flaschen[17].Aktiv
        p2738717112: (vis_Ablauf.Flaschen[17].PY -120)*vis_Ablauf.Flaschen[17].Aktiv
        tap vis_Ablauf.Taster_Flasche[17]
        Ellipse (0,0 50x50)
        Ellipse (5,5 40x40)
    Group (370,710 50x50)
        p3560616238: (vis_Ablauf.Flaschen[27].PX -300)*vis_Ablauf.Flaschen[27].Aktiv
        p2738717112: (vis_Ablauf.Flaschen[27].PY -170)*vis_Ablauf.Flaschen[27].Aktiv
        tap vis_Ablauf.Taster_Flasche[27]
        Ellipse (0,0 50x50)
            tap vis_Ablauf.Taster_Flasche[20]
        Ellipse (12,12 26x26)
    Group (420,710 50x50)
        p3560616238: (vis_Ablauf.Flaschen[28].PX -350)*vis_Ablauf.Flaschen[28].Aktiv
        p2738717112: (vis_Ablauf.Flaschen[28].PY -170)*vis_Ablauf.Flaschen[28].Aktiv
        tap vis_Ablauf.Taster_Flasche[28]
        Ellipse (0,0 50x50)
            tap vis_Ablauf.Taster_Flasche[20]
        Ellipse (12,12 26x26)
    Group (370,760 50x50)
        p3560616238: (vis_Ablauf.Flaschen[37].PX - 300 )*vis_Ablauf.Flaschen[37].Aktiv
        p2738717112: (vis_Ablauf.Flaschen[37].PY -220)*vis_Ablauf.Flaschen[37].Aktiv
        tap vis_Ablauf.Taster_Flasche[37]
        Ellipse (0,0 50x50)
        Ellipse (5,5 40x40)
    Group (420,760 50x50)
        p3560616238: (vis_Ablauf.Flaschen[38].PX - 350 )*vis_Ablauf.Flaschen[38].Aktiv
        p2738717112: (vis_Ablauf.Flaschen[38].PY -220)*vis_Ablauf.Flaschen[38].Aktiv
        tap vis_Ablauf.Taster_Flasche[38]
        Ellipse (0,0 50x50)
        Ellipse (5,5 40x40)
    Rectangle (550,715 161x105)
    Ellipse (635,740 70x70)
    Ellipse (556,740 70x70)
    Ellipse (561,745 60x60), colour toggle: vis_Ablauf.M_Init_Stellung
        tap vis_Ablauf.M_Init_Stellung
    Label (556,710 70x30), "Init Stellung"
    Ellipse (640,745 60x60), colour toggle: vis_Ablauf.M_Init_Testcase
        tap vis_Ablauf.M_Init_Testcase
    Label (635,710 70x30), "Init Testcase"
END_VISUALIZATION
